REGION Network 33: **** 2.2 - Alarms - Alarms Generation **** Fuse Locc-Box Short circuit Alarm (Condition)
   // Condition for the Alarm
   #AlarmCondShortCirc := #FuseState_BitShortCirc AND #I_EnableAlarm AND NOT #C_LevelShortCirc;
END_REGION

REGION Network 34: **** 2.2 - Alarms - Alarms Generation **** Fuse Locc-Box Short circuit Alarm
   // Memorisation of the Alarm
   IF (#I_AlarmResetPB AND NOT #C_LocalResetShortCirc) OR NOT #I_EnableAlarm OR #HMICmdResetShortCirc THEN
       #AlarmShortCirc := FALSE;   // RS flip-flop
   END_IF;
   IF #AlarmCondShortCirc THEN #AlarmShortCirc := TRUE; END_IF;
END_REGION

REGION Network 35: **** 2.2 - Alarms - Alarms Generation **** Fuse Locc-Box Short circuit Warning
   // Memorisation of the Alarm
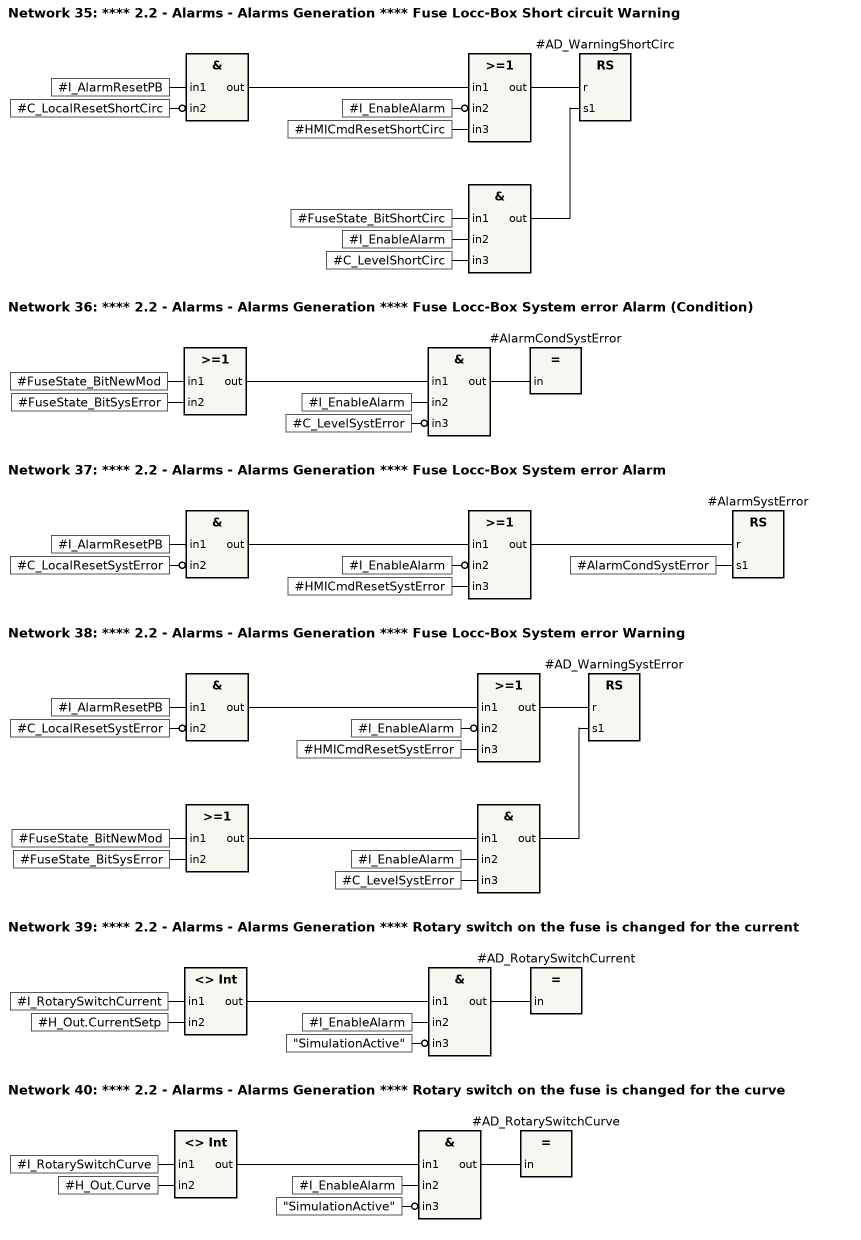
   IF (#I_AlarmResetPB AND NOT #C_LocalResetShortCirc) OR NOT #I_EnableAlarm OR #HMICmdResetShortCirc THEN
       #AD_WarningShortCirc := FALSE;   // RS flip-flop
   END_IF;
   IF #FuseState_BitShortCirc AND #I_EnableAlarm AND #C_LevelShortCirc THEN
       #AD_WarningShortCirc := TRUE;
   END_IF;
END_REGION

REGION Network 36: **** 2.2 - Alarms - Alarms Generation **** Fuse Locc-Box System error Alarm (Condition)
   // Condition for the Alarm
   #AlarmCondSystError := (#FuseState_BitNewMod OR #FuseState_BitSysError) AND #I_EnableAlarm AND NOT #C_LevelSystError;
END_REGION

REGION Network 37: **** 2.2 - Alarms - Alarms Generation **** Fuse Locc-Box System error Alarm
   // Memorisation of the Alarm
   IF (#I_AlarmResetPB AND NOT #C_LocalResetSystError) OR NOT #I_EnableAlarm OR #HMICmdResetSystError THEN
       #AlarmSystError := FALSE;   // RS flip-flop
   END_IF;
   IF #AlarmCondSystError THEN #AlarmSystError := TRUE; END_IF;
END_REGION

REGION Network 38: **** 2.2 - Alarms - Alarms Generation **** Fuse Locc-Box System error Warning
   // Memorisation of the Alarm
   IF (#I_AlarmResetPB AND NOT #C_LocalResetSystError) OR NOT #I_EnableAlarm OR #HMICmdResetSystError THEN
       #AD_WarningSystError := FALSE;   // RS flip-flop
   END_IF;
   IF (#FuseState_BitNewMod OR #FuseState_BitSysError) AND #I_EnableAlarm AND #C_LevelSystError THEN
       #AD_WarningSystError := TRUE;
   END_IF;
END_REGION

REGION Network 39: **** 2.2 - Alarms - Alarms Generation **** Rotary switch on the fuse is changed for the current
   // Alarm
   #AD_RotarySwitchCurrent := (#I_RotarySwitchCurrent <> #H_Out.CurrentSetp) AND #I_EnableAlarm AND NOT "SimulationActive";
END_REGION

REGION Network 40: **** 2.2 - Alarms - Alarms Generation **** Rotary switch on the fuse is changed for the curve
   // Alarm
   #AD_RotarySwitchCurve := (#I_RotarySwitchCurve <> #H_Out.Curve) AND #I_EnableAlarm AND NOT "SimulationActive";
END_REGION

REGION Network 41: **** 2.2 - Alarms - Alarms Generation **** Alarm = Class 'A'
   // Alarm = Class 'A'
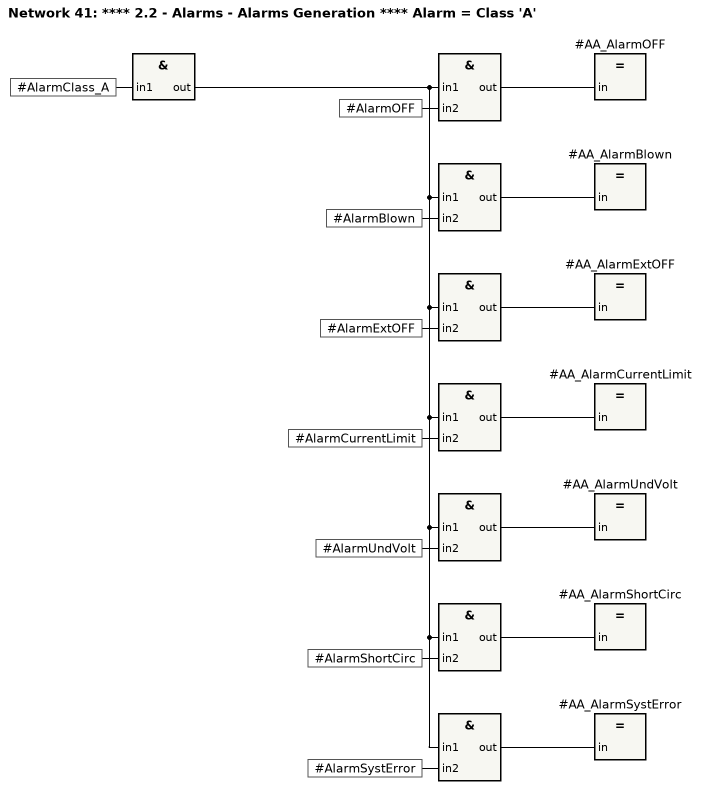
   #AA_AlarmOFF := #AlarmClass_A AND #AlarmOFF;
   #AA_AlarmBlown := #AlarmClass_A AND #AlarmBlown;
   #AA_AlarmExtOFF := #AlarmClass_A AND #AlarmExtOFF;
   #AA_AlarmCurrentLimit := #AlarmClass_A AND #AlarmCurrentLimit;
   #AA_AlarmUndVolt := #AlarmClass_A AND #AlarmUndVolt;
   #AA_AlarmShortCirc := #AlarmClass_A AND #AlarmShortCirc;
   #AA_AlarmSystError := #AlarmClass_A AND #AlarmSystError;
END_REGION

REGION Network 42: **** 2.2 - Alarms - Alarms Generation **** Alarm = Class 'B'
   // Alarm = Class 'B'
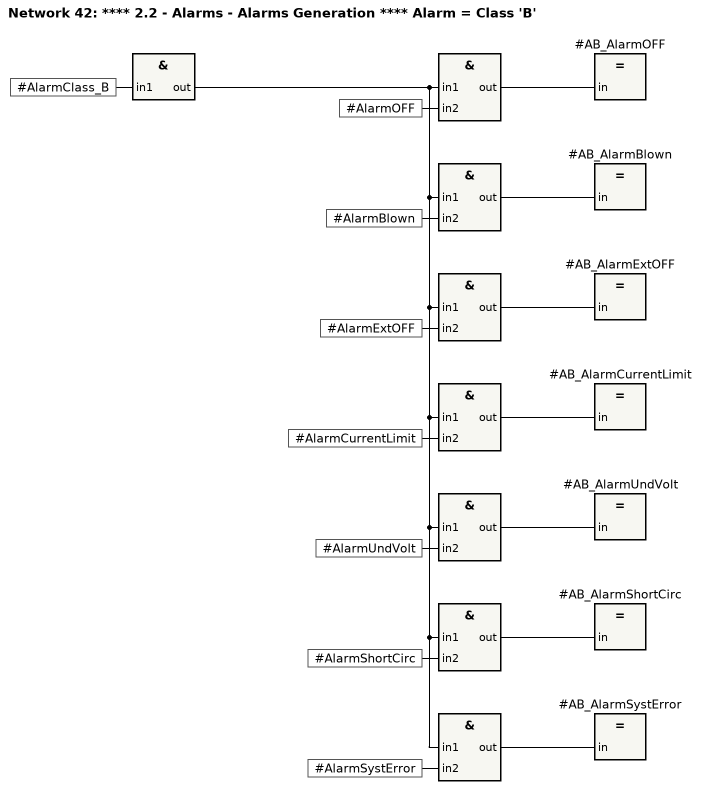
   #AB_AlarmOFF := #AlarmClass_B AND #AlarmOFF;
   #AB_AlarmBlown := #AlarmClass_B AND #AlarmBlown;
   #AB_AlarmExtOFF := #AlarmClass_B AND #AlarmExtOFF;
   #AB_AlarmCurrentLimit := #AlarmClass_B AND #AlarmCurrentLimit;
   #AB_AlarmUndVolt := #AlarmClass_B AND #AlarmUndVolt;
   #AB_AlarmShortCirc := #AlarmClass_B AND #AlarmShortCirc;
   #AB_AlarmSystError := #AlarmClass_B AND #AlarmSystError;
END_REGION

REGION Network 43: **** 2.2 - Alarms - Alarms Generation **** Alarm = Class 'C'
   // Alarm = Class 'C'
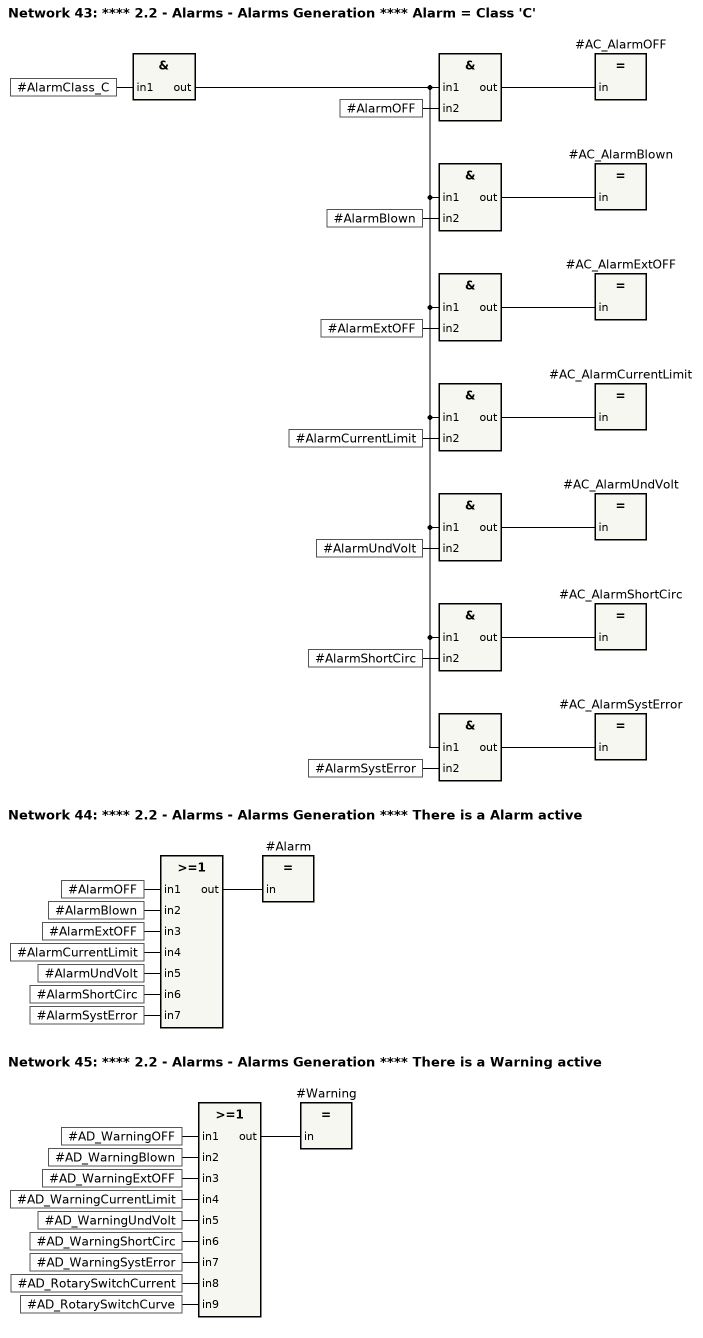
   #AC_AlarmOFF := #AlarmClass_C AND #AlarmOFF;
   #AC_AlarmBlown := #AlarmClass_C AND #AlarmBlown;
   #AC_AlarmExtOFF := #AlarmClass_C AND #AlarmExtOFF;
   #AC_AlarmCurrentLimit := #AlarmClass_C AND #AlarmCurrentLimit;
   #AC_AlarmUndVolt := #AlarmClass_C AND #AlarmUndVolt;
   #AC_AlarmShortCirc := #AlarmClass_C AND #AlarmShortCirc;
   #AC_AlarmSystError := #AlarmClass_C AND #AlarmSystError;
END_REGION

REGION Network 44: **** 2.2 - Alarms - Alarms Generation **** There is a Alarm active
   // There is a Alarm active
   #Alarm := #AlarmOFF OR #AlarmBlown OR #AlarmExtOFF OR #AlarmCurrentLimit OR #AlarmUndVolt OR #AlarmShortCirc OR #AlarmSystError;
END_REGION

REGION Network 45: **** 2.2 - Alarms - Alarms Generation **** There is a Warning active
   // There is a Warning active
   #Warning := #AD_WarningOFF OR #AD_WarningBlown OR #AD_WarningExtOFF OR #AD_WarningCurrentLimit OR #AD_WarningUndVolt OR #AD_WarningShortCirc OR #AD_WarningSystError OR #AD_RotarySwitchCurrent OR #AD_RotarySwitchCurve;
END_REGION

REGION Network 46: **** 3 - Communication - Other Systems **** Read info from LoccBox Fuse
   // Read info from LoccBox Fuse
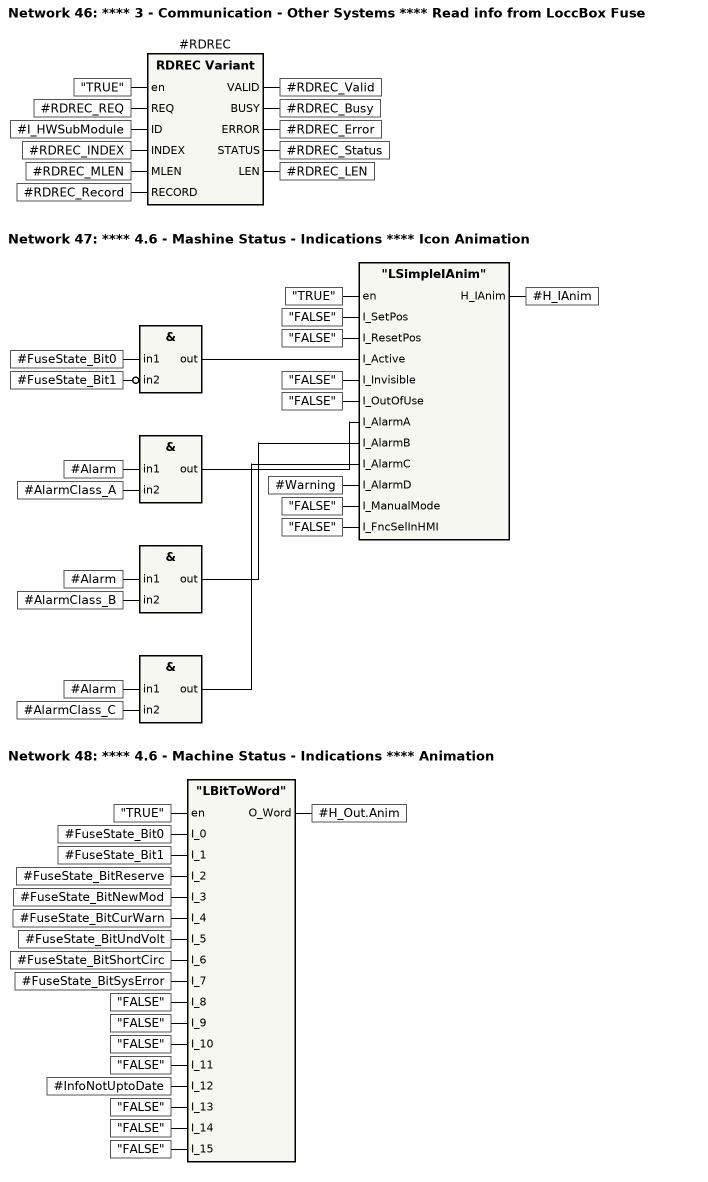
   IF "TRUE" THEN
       #RDREC(REQ := #RDREC_REQ,   // RDREC
              ID := #I_HWSubModule,
              INDEX := #RDREC_INDEX,
              MLEN := #RDREC_MLEN,
              RECORD := #RDREC_Record,
              VALID => #RDREC_Valid,
              BUSY => #RDREC_Busy,
              ERROR => #RDREC_Error,
              STATUS => #RDREC_Status,
              LEN => #RDREC_LEN);
   END_IF;
END_REGION

REGION Network 47: **** 4.6 - Mashine Status - Indications **** Icon Animation
   // Icon Animation
   IF "TRUE" THEN
       "LSimpleIAnim"(I_SetPos := "FALSE",
                      I_ResetPos := "FALSE",
                      I_Active := #FuseState_Bit0 AND NOT #FuseState_Bit1,
                      I_Invisible := "FALSE",
                      I_OutOfUse := "FALSE",
                      I_AlarmA := #Alarm AND #AlarmClass_A,
                      I_AlarmB := #Alarm AND #AlarmClass_B,
                      I_AlarmC := #Alarm AND #AlarmClass_C,
                      I_AlarmD := #Warning,
                      I_ManualMode := "FALSE",
                      I_FncSelInHMI := "FALSE",
                      H_IAnim => #H_IAnim);
   END_IF;
END_REGION

REGION Network 48: **** 4.6 - Machine Status - Indications **** Animation
   // Animation
   IF "TRUE" THEN
       "LBitToWord"(I_0 := #FuseState_Bit0,
                    I_1 := #FuseState_Bit1,
                    I_2 := #FuseState_BitReserve,
                    I_3 := #FuseState_BitNewMod,
                    I_4 := #FuseState_BitCurWarn,
                    I_5 := #FuseState_BitUndVolt,
                    I_6 := #FuseState_BitShortCirc,
                    I_7 := #FuseState_BitSysError,
                    I_8 := "FALSE",
                    I_9 := "FALSE",
                    I_10 := "FALSE",
                    I_11 := "FALSE",
                    I_12 := #InfoNotUptoDate,
                    I_13 := "FALSE",
                    I_14 := "FALSE",
                    I_15 := "FALSE",
                    O_Word => #H_Out.Anim);
   END_IF;
END_REGION

REGION Network 49: **** 4.6 - Machine Status - Indications **** Animation2
   // Animation
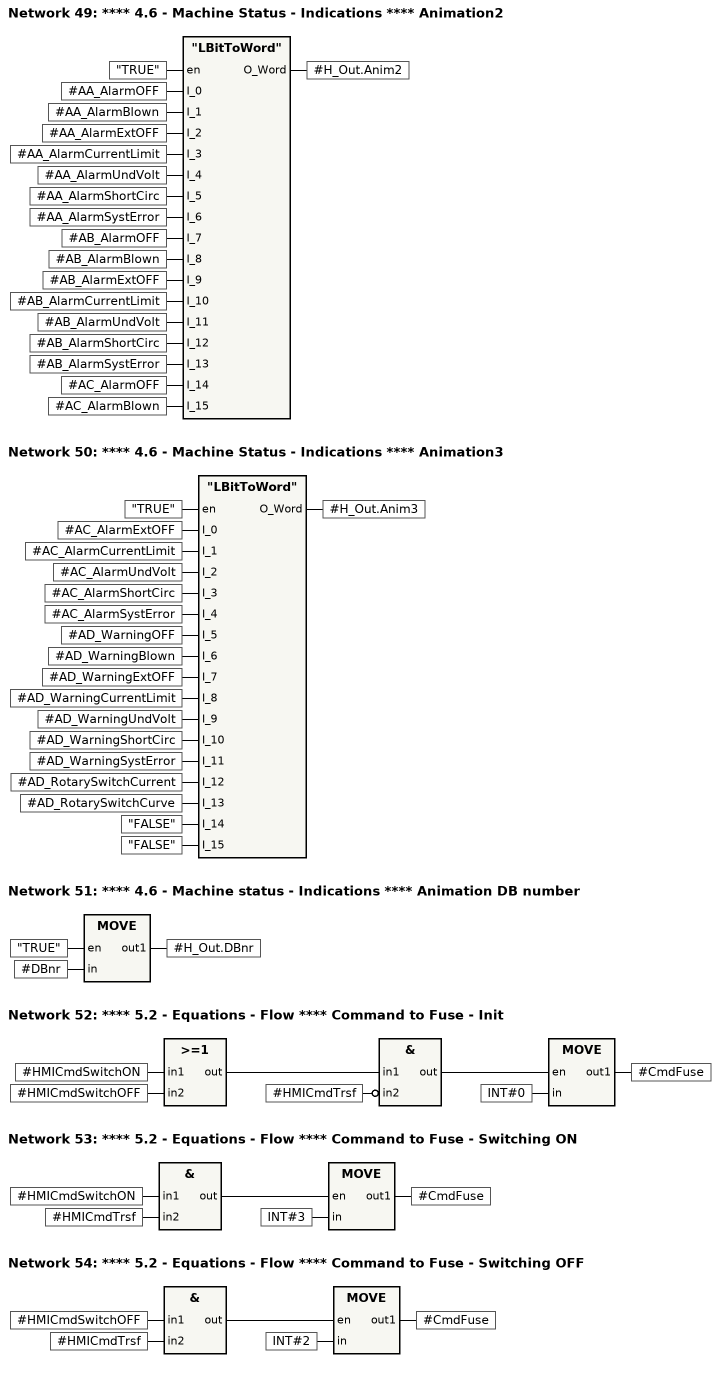
   IF "TRUE" THEN
       "LBitToWord"(I_0 := #AA_AlarmOFF,
                    I_1 := #AA_AlarmBlown,
                    I_2 := #AA_AlarmExtOFF,
                    I_3 := #AA_AlarmCurrentLimit,
                    I_4 := #AA_AlarmUndVolt,
                    I_5 := #AA_AlarmShortCirc,
                    I_6 := #AA_AlarmSystError,
                    I_7 := #AB_AlarmOFF,
                    I_8 := #AB_AlarmBlown,
                    I_9 := #AB_AlarmExtOFF,
                    I_10 := #AB_AlarmCurrentLimit,
                    I_11 := #AB_AlarmUndVolt,
                    I_12 := #AB_AlarmShortCirc,
                    I_13 := #AB_AlarmSystError,
                    I_14 := #AC_AlarmOFF,
                    I_15 := #AC_AlarmBlown,
                    O_Word => #H_Out.Anim2);
   END_IF;
END_REGION

REGION Network 50: **** 4.6 - Machine Status - Indications **** Animation3
   // Animation
   IF "TRUE" THEN
       "LBitToWord"(I_0 := #AC_AlarmExtOFF,
                    I_1 := #AC_AlarmCurrentLimit,
                    I_2 := #AC_AlarmUndVolt,
                    I_3 := #AC_AlarmShortCirc,
                    I_4 := #AC_AlarmSystError,
                    I_5 := #AD_WarningOFF,
                    I_6 := #AD_WarningBlown,
                    I_7 := #AD_WarningExtOFF,
                    I_8 := #AD_WarningCurrentLimit,
                    I_9 := #AD_WarningUndVolt,
                    I_10 := #AD_WarningShortCirc,
                    I_11 := #AD_WarningSystError,
                    I_12 := #AD_RotarySwitchCurrent,
                    I_13 := #AD_RotarySwitchCurve,
                    I_14 := "FALSE",
                    I_15 := "FALSE",
                    O_Word => #H_Out.Anim3);
   END_IF;
END_REGION

REGION Network 51: **** 4.6 - Machine status - Indications **** Animation DB number
   // DB number
   IF "TRUE" THEN #H_Out.DBnr := #DBnr; END_IF;
END_REGION

REGION Network 52: **** 5.2 - Equations - Flow **** Command to Fuse - Init
   // Write zero to outputbyte to have an transition from 0 to ...
   IF (#HMICmdSwitchON OR #HMICmdSwitchOFF) AND NOT #HMICmdTrsf THEN #CmdFuse := INT#0; END_IF;
END_REGION

REGION Network 53: **** 5.2 - Equations - Flow **** Command to Fuse - Switching ON
   // Switching ON
   IF #HMICmdSwitchON AND #HMICmdTrsf THEN #CmdFuse := INT#3; END_IF;
END_REGION

REGION Network 54: **** 5.2 - Equations - Flow **** Command to Fuse - Switching OFF
   // Switching OFF
   IF #HMICmdSwitchOFF AND #HMICmdTrsf THEN #CmdFuse := INT#2; END_IF;
END_REGION

REGION Network 55: **** 5.2 - Equations - Flow **** Start Read function (GET Info)
   // Start Read function
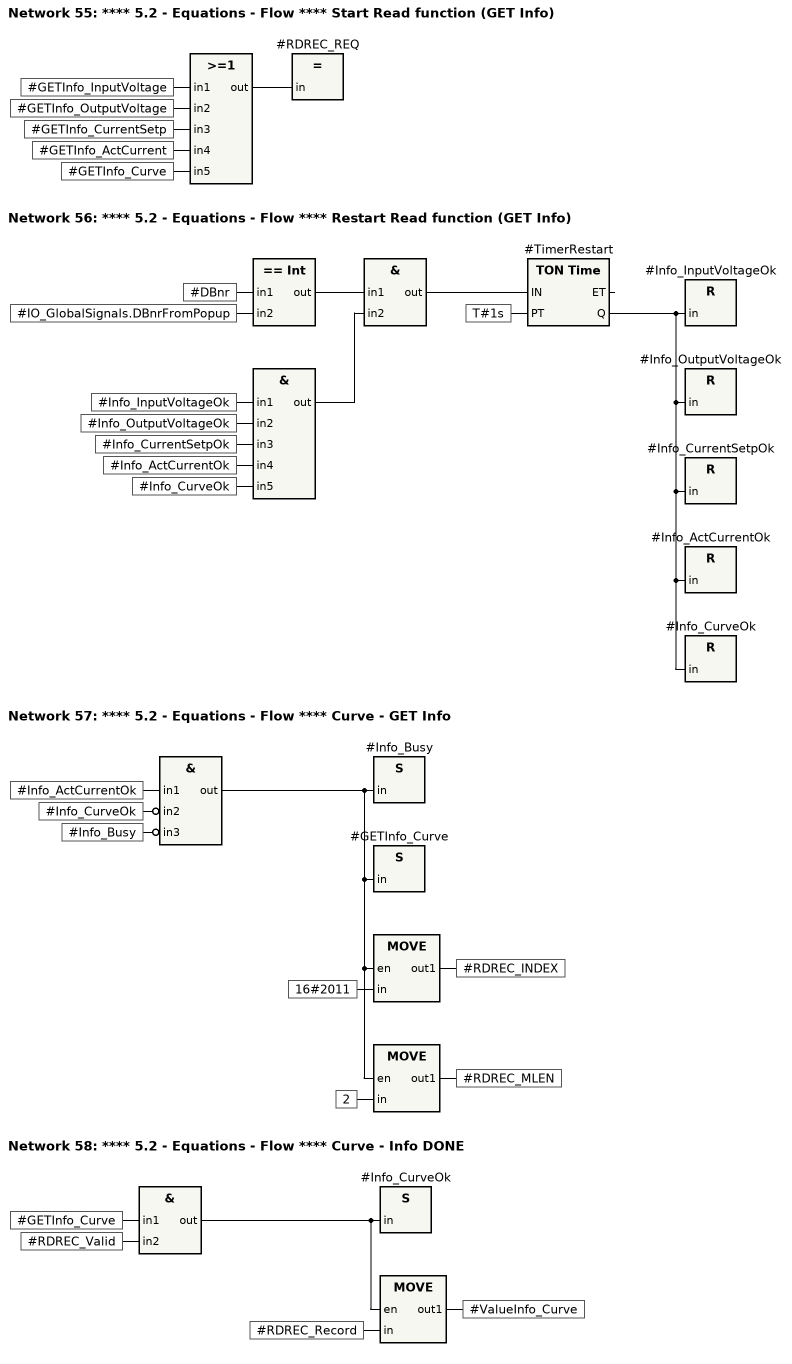
   #RDREC_REQ := #GETInfo_InputVoltage OR #GETInfo_OutputVoltage OR #GETInfo_CurrentSetp OR #GETInfo_ActCurrent OR #GETInfo_Curve;
END_REGION

REGION Network 56: **** 5.2 - Equations - Flow **** Restart Read function (GET Info)
   // Restart Read function (GET Info)
   #TimerRestart(IN := (#DBnr = #IO_GlobalSignals.DBnrFromPopup) AND #Info_InputVoltageOk AND #Info_OutputVoltageOk AND #Info_CurrentSetpOk AND #Info_ActCurrentOk AND #Info_CurveOk,   // TON
                 PT := T#1s);
   IF #TimerRestart.Q THEN
       #Info_InputVoltageOk := FALSE;
       #Info_OutputVoltageOk := FALSE;
       #Info_CurrentSetpOk := FALSE;
       #Info_ActCurrentOk := FALSE;
       #Info_CurveOk := FALSE;
   END_IF;
END_REGION

REGION Network 57: **** 5.2 - Equations - Flow **** Curve - GET Info
   // GET Info Curve
   #_w1 := #Info_ActCurrentOk AND NOT #Info_CurveOk AND NOT #Info_Busy;
   IF #_w1 THEN
       #Info_Busy := TRUE;
       #GETInfo_Curve := TRUE;
       #RDREC_INDEX := 16#2011;
       #RDREC_MLEN := 2;
   END_IF;
END_REGION

REGION Network 58: **** 5.2 - Equations - Flow **** Curve - Info DONE
   // DONE Info Curve
   IF #GETInfo_Curve AND #RDREC_Valid THEN
       #Info_CurveOk := TRUE;
       #ValueInfo_Curve := #RDREC_Record;
   END_IF;
END_REGION

REGION Network 59: **** 5.2 - Equations - Flow **** Curve - CALCULATE
   // CALCULATE Current Curve
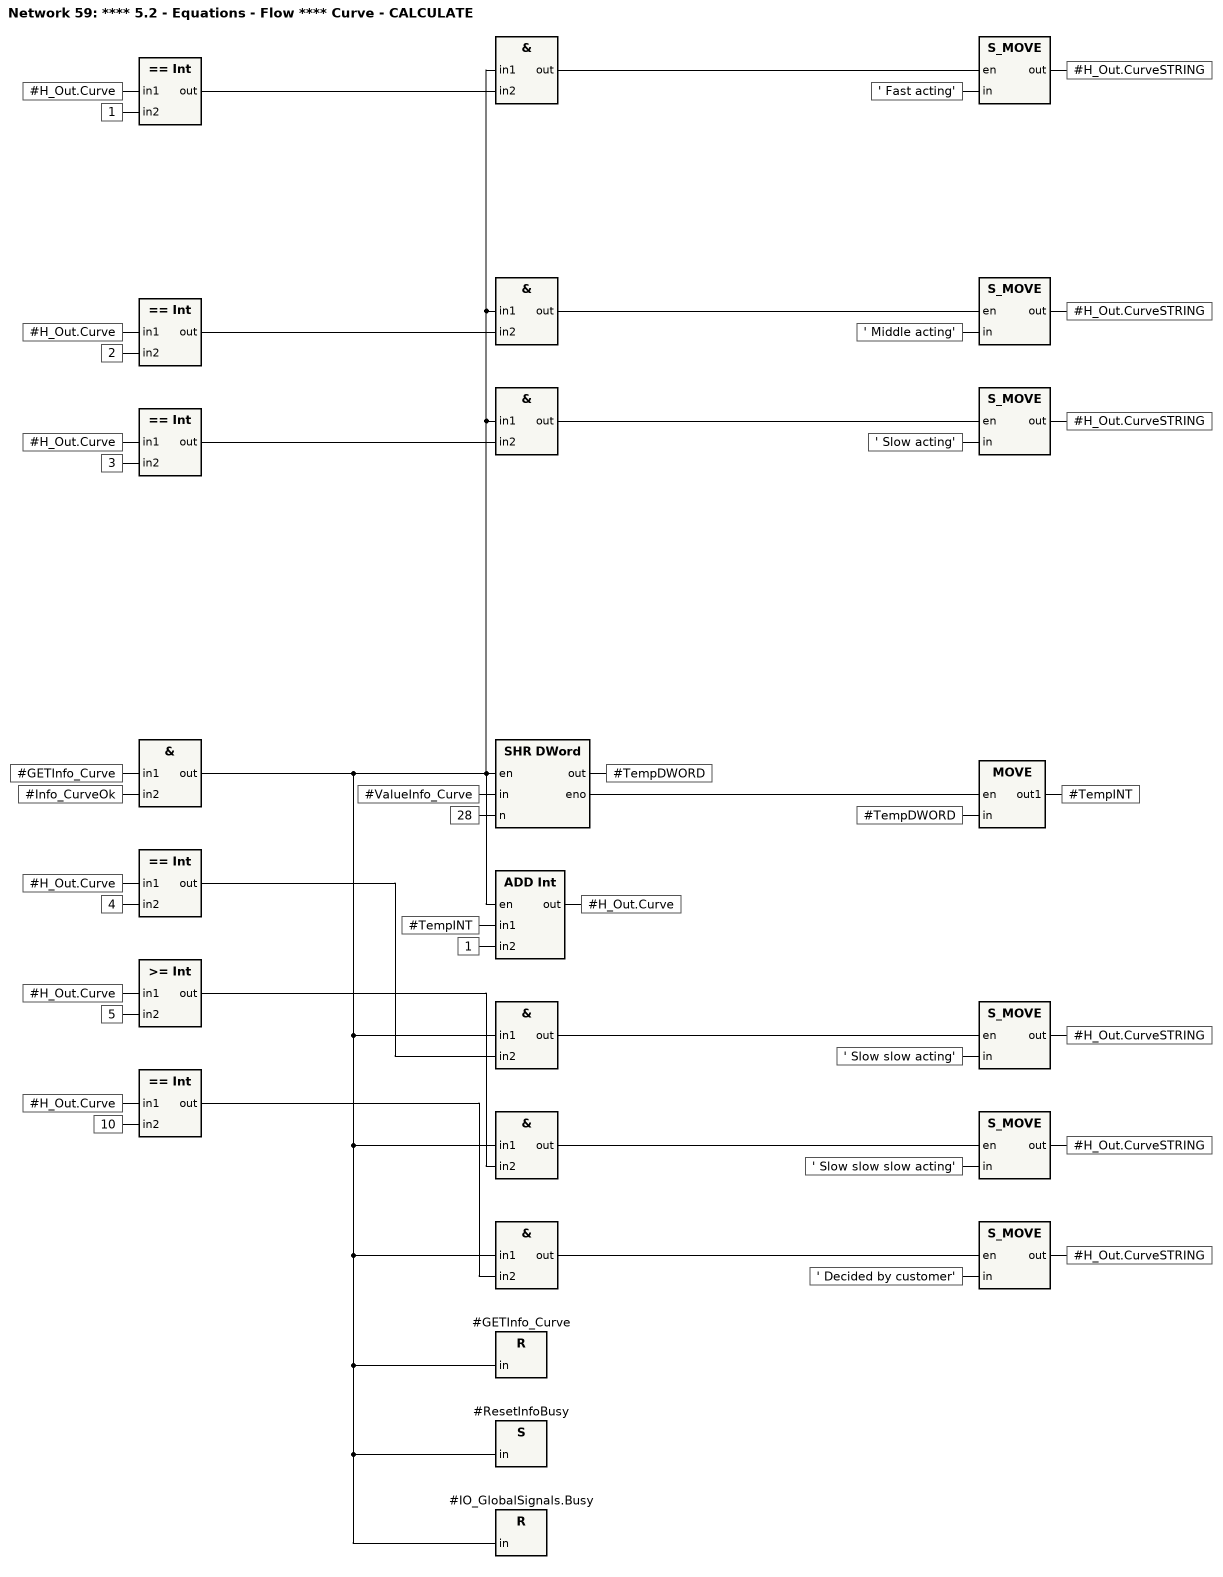
   #_w1 := #GETInfo_Curve AND #Info_CurveOk;
   IF #_w1 THEN
       #TempDWORD := SHR(IN := #ValueInfo_Curve, N := 28);
       #TempINT := #TempDWORD;
       #H_Out.Curve := #TempINT + 1;
   END_IF;
   IF #_w1 AND (#H_Out.Curve = 1) THEN #H_Out.CurveSTRING := ' Fast acting'; END_IF;
   IF #_w1 AND (#H_Out.Curve = 2) THEN #H_Out.CurveSTRING := ' Middle acting'; END_IF;
   IF #_w1 AND (#H_Out.Curve = 3) THEN #H_Out.CurveSTRING := ' Slow acting'; END_IF;
   IF #_w1 AND (#H_Out.Curve = 4) THEN #H_Out.CurveSTRING := ' Slow slow acting'; END_IF;
   IF #_w1 AND (#H_Out.Curve >= 5) THEN #H_Out.CurveSTRING := ' Slow slow slow acting'; END_IF;
   IF #_w1 AND (#H_Out.Curve = 10) THEN #H_Out.CurveSTRING := ' Decided by customer'; END_IF;
   IF #_w1 THEN
       #GETInfo_Curve := FALSE;
       #ResetInfoBusy := TRUE;
       #IO_GlobalSignals.Busy := FALSE;
   END_IF;
END_REGION

REGION Network 60: **** 5.2 - Equations - Flow **** Actual Current - GET Info
   // GET Info Actual Current
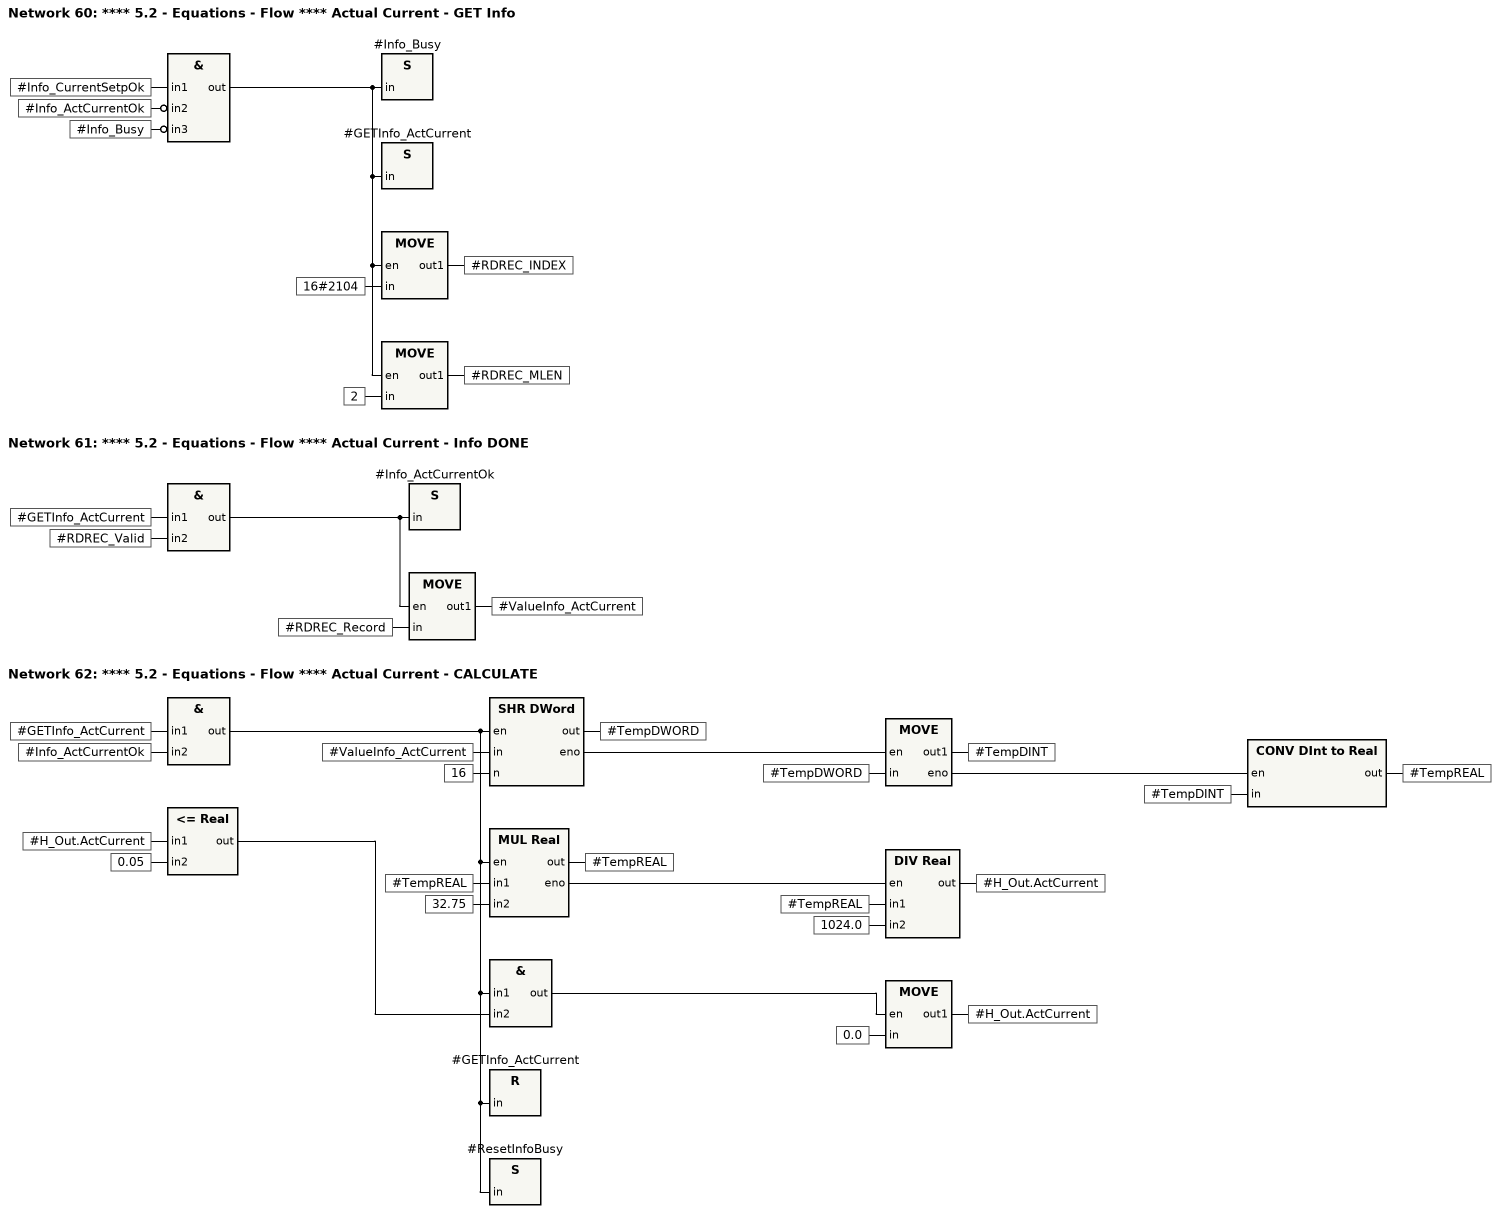
   #_w1 := #Info_CurrentSetpOk AND NOT #Info_ActCurrentOk AND NOT #Info_Busy;
   IF #_w1 THEN
       #Info_Busy := TRUE;
       #GETInfo_ActCurrent := TRUE;
       #RDREC_INDEX := 16#2104;
       #RDREC_MLEN := 2;
   END_IF;
END_REGION

REGION Network 61: **** 5.2 - Equations - Flow **** Actual Current - Info DONE
   // DONE Info Actual Current
   IF #GETInfo_ActCurrent AND #RDREC_Valid THEN
       #Info_ActCurrentOk := TRUE;
       #ValueInfo_ActCurrent := #RDREC_Record;
   END_IF;
END_REGION

REGION Network 62: **** 5.2 - Equations - Flow **** Actual Current - CALCULATE
   // CALCULATE Actual Current   ----->  Actual Current = (ValueInfo_ActCurrent * 32,75A) / 1024
   #_w1 := #GETInfo_ActCurrent AND #Info_ActCurrentOk;
   IF #_w1 THEN
       #TempDWORD := SHR(IN := #ValueInfo_ActCurrent, N := 16);
       #TempDINT := #TempDWORD;
       #TempREAL := DINT_TO_REAL(#TempDINT);
       #TempREAL := #TempREAL * 32.75;
       #H_Out.ActCurrent := #TempREAL / 1024.0;
   END_IF;
   IF #_w1 AND (#H_Out.ActCurrent <= 0.05) THEN #H_Out.ActCurrent := 0.0; END_IF;
   IF #_w1 THEN
       #GETInfo_ActCurrent := FALSE;
       #ResetInfoBusy := TRUE;
   END_IF;
END_REGION

REGION Network 63: **** 5.2 - Equations - Flow **** Current Setpoint - GET Info
   // GET Info Current Setpoint
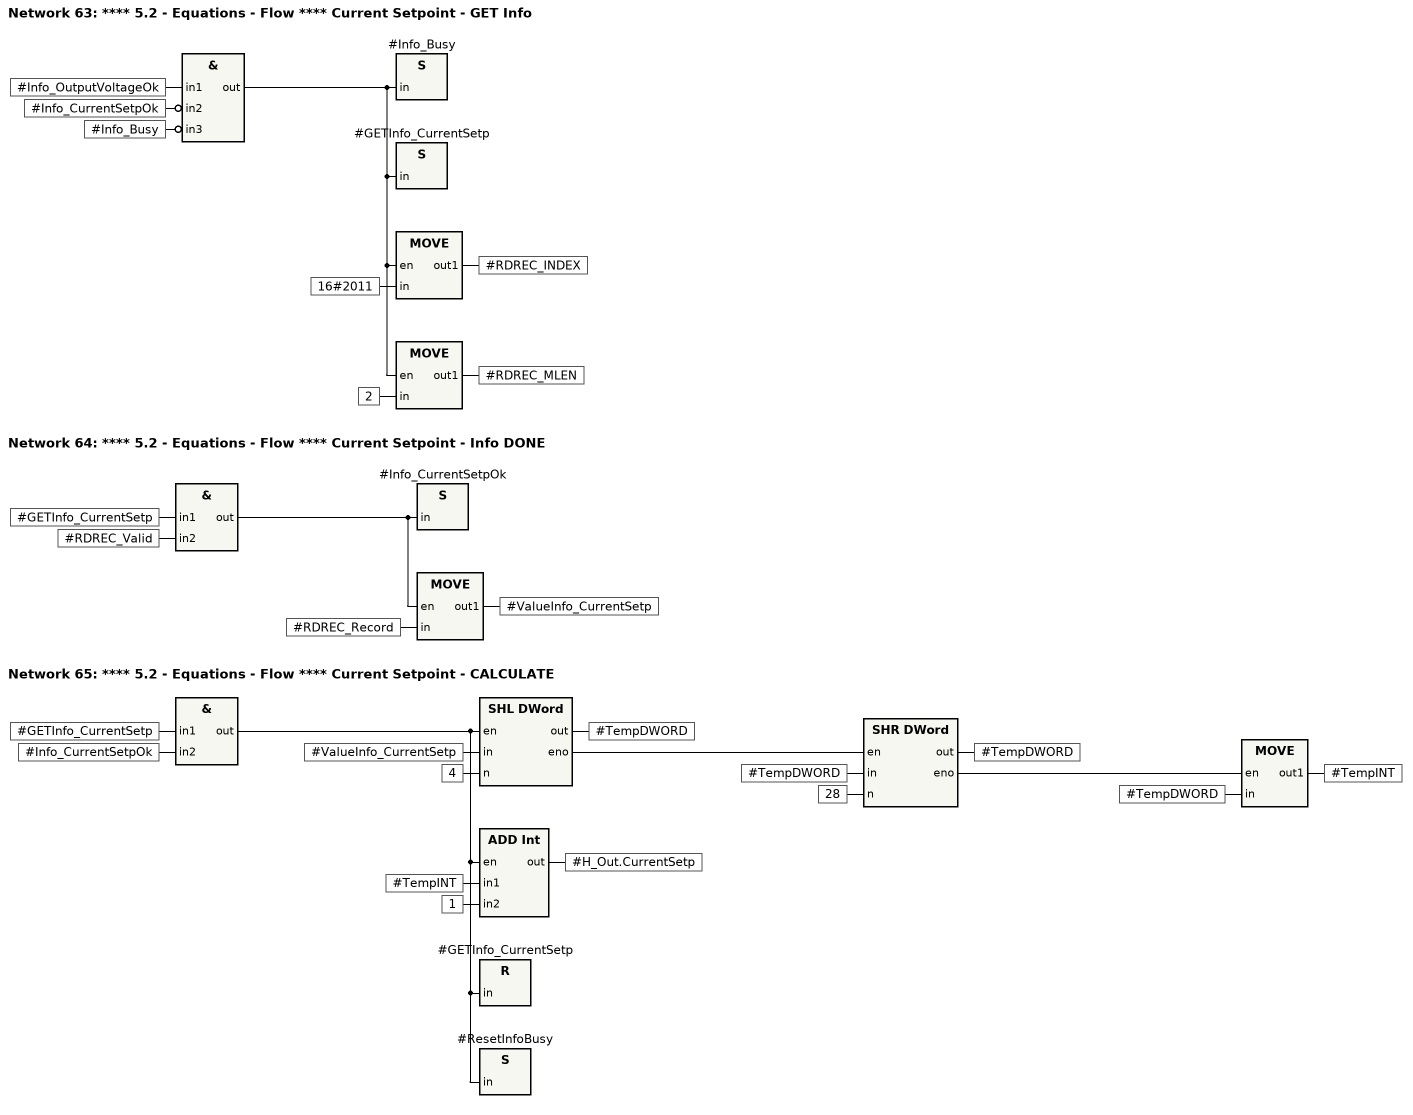
   #_w1 := #Info_OutputVoltageOk AND NOT #Info_CurrentSetpOk AND NOT #Info_Busy;
   IF #_w1 THEN
       #Info_Busy := TRUE;
       #GETInfo_CurrentSetp := TRUE;
       #RDREC_INDEX := 16#2011;
       #RDREC_MLEN := 2;
   END_IF;
END_REGION

REGION Network 64: **** 5.2 - Equations - Flow **** Current Setpoint - Info DONE
   // DONE Info Current Setpoint
   IF #GETInfo_CurrentSetp AND #RDREC_Valid THEN
       #Info_CurrentSetpOk := TRUE;
       #ValueInfo_CurrentSetp := #RDREC_Record;
   END_IF;
END_REGION

REGION Network 65: **** 5.2 - Equations - Flow **** Current Setpoint - CALCULATE
   // CALCULATE Current Setpoint
   IF #GETInfo_CurrentSetp AND #Info_CurrentSetpOk THEN
       #TempDWORD := SHL(IN := #ValueInfo_CurrentSetp, N := 4);
       #TempDWORD := SHR(IN := #TempDWORD, N := 28);
       #TempINT := #TempDWORD;
       #H_Out.CurrentSetp := #TempINT + 1;
   END_IF;
   #_w1 := #GETInfo_CurrentSetp AND #Info_CurrentSetpOk;
   IF #_w1 THEN
       #GETInfo_CurrentSetp := FALSE;
       #ResetInfoBusy := TRUE;
   END_IF;
END_REGION

REGION Network 66: **** 5.2 - Equations - Flow **** Output Voltage - GET Info
   // GET Info Output Voltage
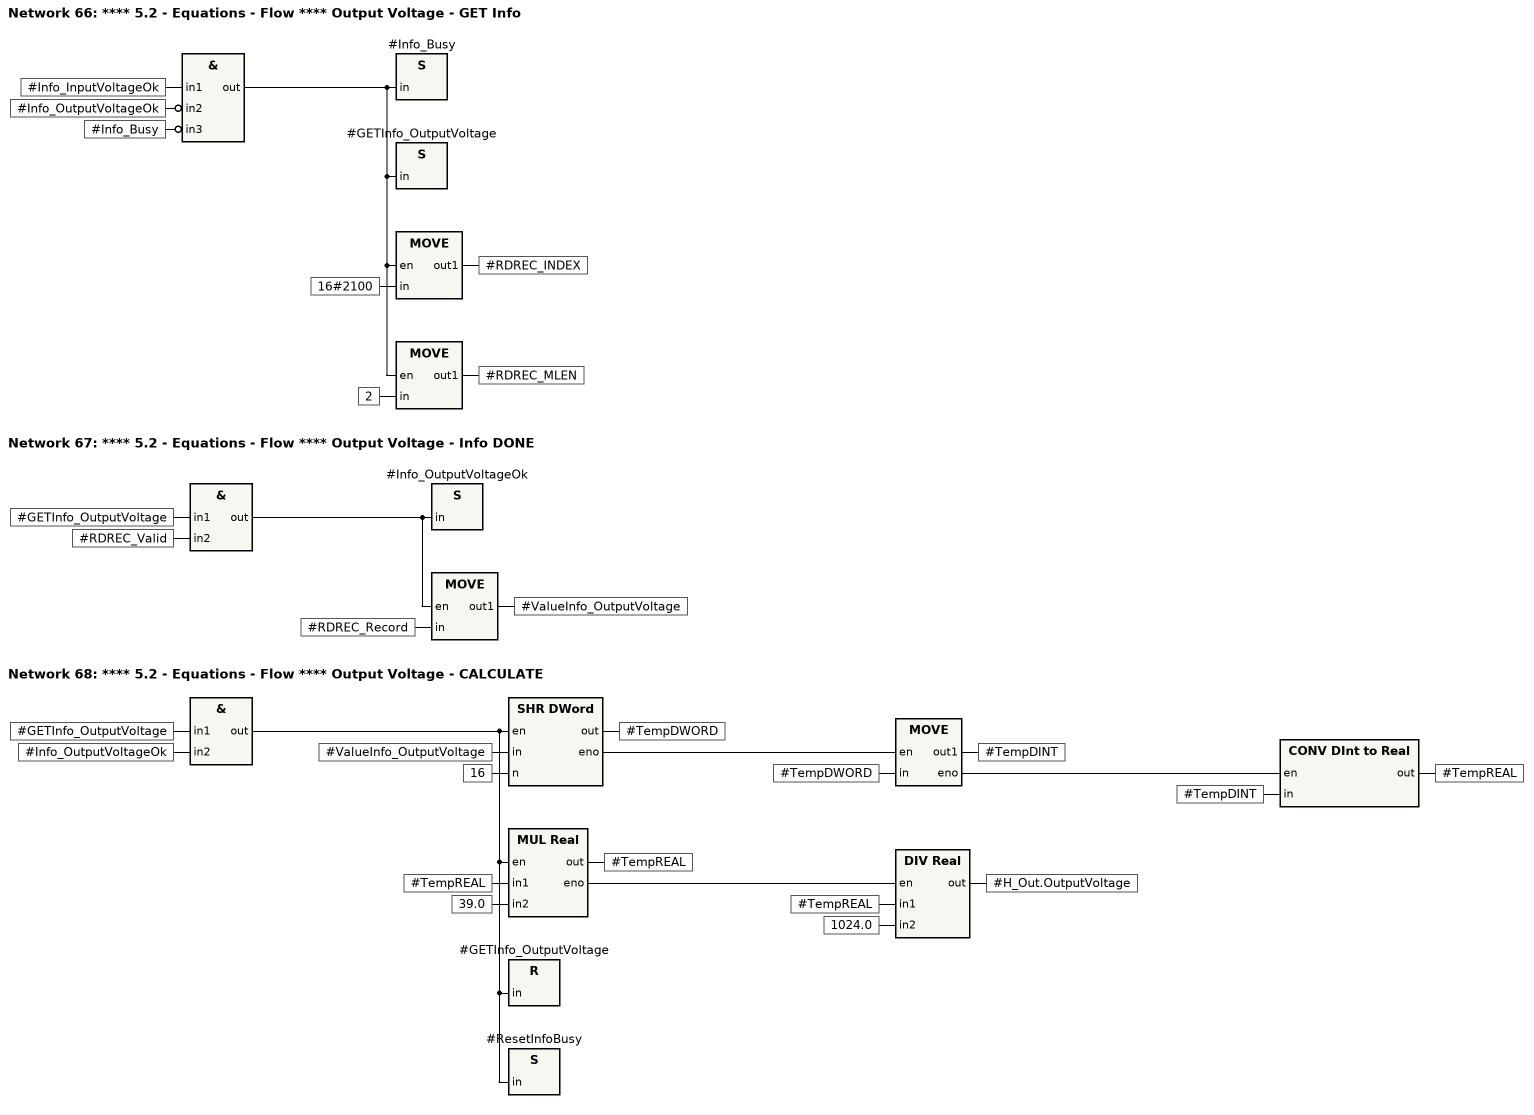
   #_w1 := #Info_InputVoltageOk AND NOT #Info_OutputVoltageOk AND NOT #Info_Busy;
   IF #_w1 THEN
       #Info_Busy := TRUE;
       #GETInfo_OutputVoltage := TRUE;
       #RDREC_INDEX := 16#2100;
       #RDREC_MLEN := 2;
   END_IF;
END_REGION

REGION Network 67: **** 5.2 - Equations - Flow **** Output Voltage - Info DONE
   // DONE Info Output Voltage
   IF #GETInfo_OutputVoltage AND #RDREC_Valid THEN
       #Info_OutputVoltageOk := TRUE;
       #ValueInfo_OutputVoltage := #RDREC_Record;
   END_IF;
END_REGION

REGION Network 68: **** 5.2 - Equations - Flow **** Output Voltage - CALCULATE
   // CALCULATE Output Voltage   ----->  Output Voltage = (ValueInfo_OutputVoltage * 39V) / 1024
   IF #GETInfo_OutputVoltage AND #Info_OutputVoltageOk THEN
       #TempDWORD := SHR(IN := #ValueInfo_OutputVoltage, N := 16);
       #TempDINT := #TempDWORD;
       #TempREAL := DINT_TO_REAL(#TempDINT);
       #TempREAL := #TempREAL * 39.0;
       #H_Out.OutputVoltage := #TempREAL / 1024.0;
   END_IF;
   #_w1 := #GETInfo_OutputVoltage AND #Info_OutputVoltageOk;
   IF #_w1 THEN
       #GETInfo_OutputVoltage := FALSE;
       #ResetInfoBusy := TRUE;
   END_IF;
END_REGION

REGION Network 69: **** 5.2 - Equations - Flow **** Input Voltage - GET Info
   // GET Info Input Voltage
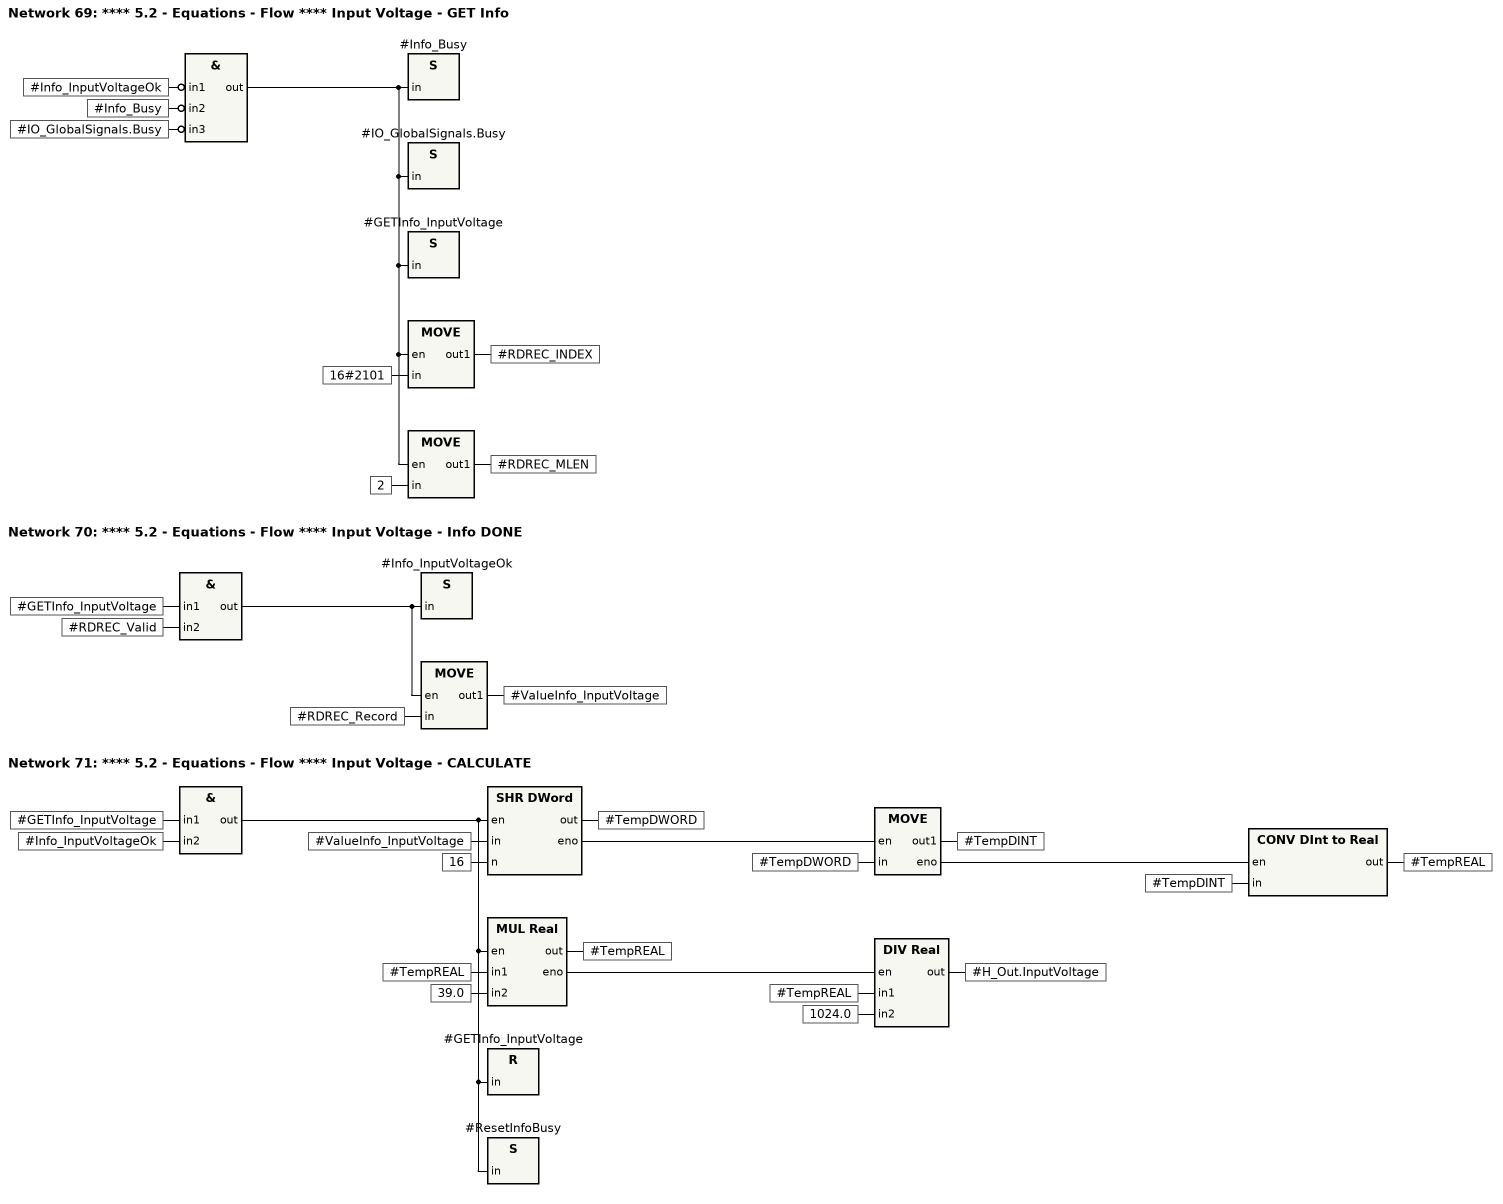
   #_w1 := NOT #Info_InputVoltageOk AND NOT #Info_Busy AND NOT #IO_GlobalSignals.Busy;
   IF #_w1 THEN
       #Info_Busy := TRUE;
       #IO_GlobalSignals.Busy := TRUE;
       #GETInfo_InputVoltage := TRUE;
       #RDREC_INDEX := 16#2101;
       #RDREC_MLEN := 2;
   END_IF;
END_REGION

REGION Network 70: **** 5.2 - Equations - Flow **** Input Voltage - Info DONE
   // DONE Info Input Voltage
   IF #GETInfo_InputVoltage AND #RDREC_Valid THEN
       #Info_InputVoltageOk := TRUE;
       #ValueInfo_InputVoltage := #RDREC_Record;
   END_IF;
END_REGION

REGION Network 71: **** 5.2 - Equations - Flow **** Input Voltage - CALCULATE
   // CALCULATE Input Voltage   ----->  Input Voltage = (ValueInfo_InputVoltage * 39V) / 1024
   IF #GETInfo_InputVoltage AND #Info_InputVoltageOk THEN
       #TempDWORD := SHR(IN := #ValueInfo_InputVoltage, N := 16);
       #TempDINT := #TempDWORD;
       #TempREAL := DINT_TO_REAL(#TempDINT);
       #TempREAL := #TempREAL * 39.0;
       #H_Out.InputVoltage := #TempREAL / 1024.0;
   END_IF;
   #_w1 := #GETInfo_InputVoltage AND #Info_InputVoltageOk;
   IF #_w1 THEN
       #GETInfo_InputVoltage := FALSE;
       #ResetInfoBusy := TRUE;
   END_IF;
END_REGION

REGION Network 72: **** 5.2 - Equations - Flow **** Local Busy
   // Local Busy
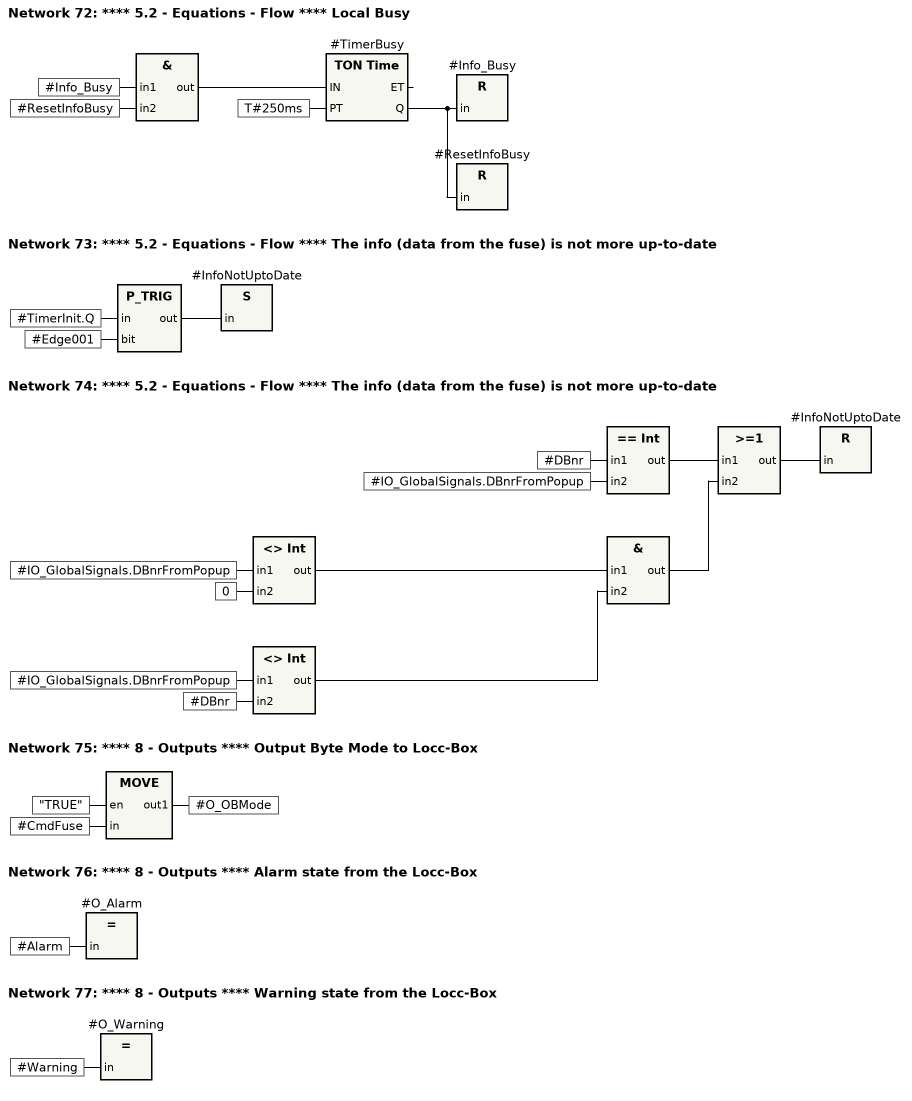
   #TimerBusy(IN := #Info_Busy AND #ResetInfoBusy, PT := T#250ms);   // TON
   IF #TimerBusy.Q THEN
       #Info_Busy := FALSE;
       #ResetInfoBusy := FALSE;
   END_IF;
END_REGION

REGION Network 73: **** 5.2 - Equations - Flow **** The info (data from the fuse) is not more up-to-date
   // The info (data from the fuse) is not more up-to-date
   #_w1 := #TimerInit.Q AND NOT #Edge001;   // rising edge
   #Edge001 := #TimerInit.Q;
   IF #_w1 THEN #InfoNotUptoDate := TRUE; END_IF;
END_REGION

REGION Network 74: **** 5.2 - Equations - Flow **** The info (data from the fuse) is not more up-to-date
   // The info (data from the fuse) is not more up-to-date
   IF (#DBnr = #IO_GlobalSignals.DBnrFromPopup) OR ((#IO_GlobalSignals.DBnrFromPopup <> 0) AND (#IO_GlobalSignals.DBnrFromPopup <> #DBnr)) THEN
       #InfoNotUptoDate := FALSE;
   END_IF;
END_REGION

REGION Network 75: **** 8 - Outputs **** Output Byte Mode to Locc-Box
   // Output Byte Mode to Locc-Box
   IF "TRUE" THEN #O_OBMode := #CmdFuse; END_IF;
END_REGION

REGION Network 76: **** 8 - Outputs **** Alarm state from the Locc-Box
   // Alarm state from the Locc-Box
   #O_Alarm := #Alarm;
END_REGION

REGION Network 77: **** 8 - Outputs **** Warning state from the Locc-Box
   // Warning state from the Locc-Box
   #O_Warning := #Warning;
END_REGION

REGION Network 78: **** 8 - Outputs **** Alarm AB condition
   // Alarm AB condition
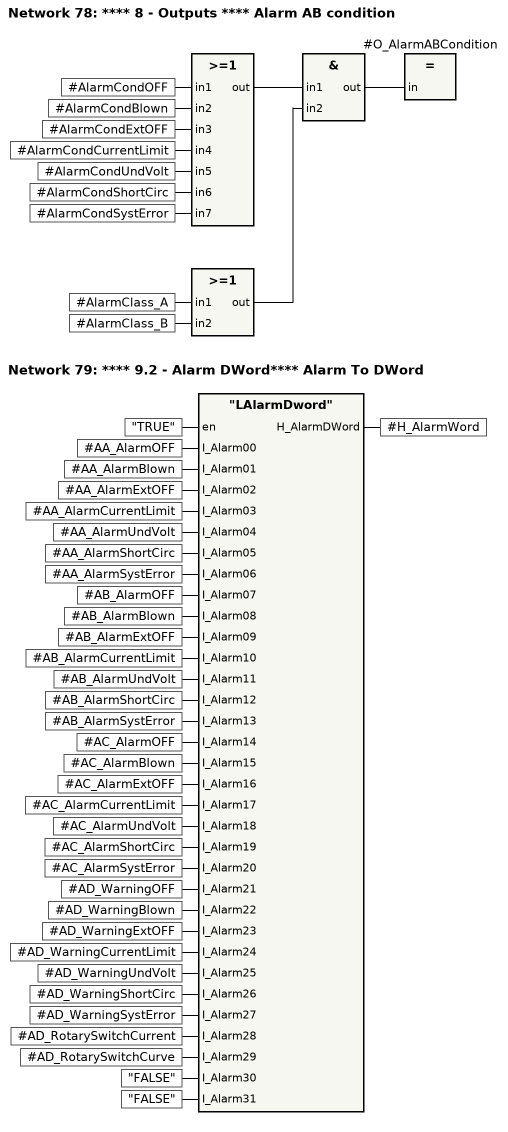
   #O_AlarmABCondition := (#AlarmCondOFF OR #AlarmCondBlown OR #AlarmCondExtOFF OR #AlarmCondCurrentLimit OR #AlarmCondUndVolt OR #AlarmCondShortCirc OR #AlarmCondSystError) AND (#AlarmClass_A OR #AlarmClass_B);
END_REGION

REGION Network 79: **** 9.2 - Alarm DWord**** Alarm To DWord
   // Alarm Word
   IF "TRUE" THEN
       "LAlarmDword"(I_Alarm00 := #AA_AlarmOFF,
                     I_Alarm01 := #AA_AlarmBlown,
                     I_Alarm02 := #AA_AlarmExtOFF,
                     I_Alarm03 := #AA_AlarmCurrentLimit,
                     I_Alarm04 := #AA_AlarmUndVolt,
                     I_Alarm05 := #AA_AlarmShortCirc,
                     I_Alarm06 := #AA_AlarmSystError,
                     I_Alarm07 := #AB_AlarmOFF,
                     I_Alarm08 := #AB_AlarmBlown,
                     I_Alarm09 := #AB_AlarmExtOFF,
                     I_Alarm10 := #AB_AlarmCurrentLimit,
                     I_Alarm11 := #AB_AlarmUndVolt,
                     I_Alarm12 := #AB_AlarmShortCirc,
                     I_Alarm13 := #AB_AlarmSystError,
                     I_Alarm14 := #AC_AlarmOFF,
                     I_Alarm15 := #AC_AlarmBlown,
                     I_Alarm16 := #AC_AlarmExtOFF,
                     I_Alarm17 := #AC_AlarmCurrentLimit,
                     I_Alarm18 := #AC_AlarmUndVolt,
                     I_Alarm19 := #AC_AlarmShortCirc,
                     I_Alarm20 := #AC_AlarmSystError,
                     I_Alarm21 := #AD_WarningOFF,
                     I_Alarm22 := #AD_WarningBlown,
                     I_Alarm23 := #AD_WarningExtOFF,
                     I_Alarm24 := #AD_WarningCurrentLimit,
                     I_Alarm25 := #AD_WarningUndVolt,
                     I_Alarm26 := #AD_WarningShortCirc,
                     I_Alarm27 := #AD_WarningSystError,
                     I_Alarm28 := #AD_RotarySwitchCurrent,
                     I_Alarm29 := #AD_RotarySwitchCurve,
                     I_Alarm30 := "FALSE",
                     I_Alarm31 := "FALSE",
                     H_AlarmDWord => #H_AlarmWord);
   END_IF;
END_REGION
END_FUNCTION_BLOCK

FUNCTION_BLOCK "LETAFuseAlarm"   // FB1413, FBD
TITLE = LLoccBoxAlarm / LETAFuseAlarm
{ S7_Optimized_Access := 'FALSE' }
AUTHOR : VCG
FAMILY : AlarmHnd
NAME : SpcGB
VERSION : 1.0
// ================================================================================
// This module is used for installations with Locc-Box type 7-6410.
// It create alarms and warning in function of configuration and status from the 
// Box.
// It Send Mode byte to the Box in function of Pop-up and external commands
// ================================================================================
// C_AlarmOrWarning
// Bit0: C_LevelOFF (Bit ON=Warning ; OFF=Alarm)
// Bit1: C_LevelBlown (Bit ON=Warning ; OFF=Alarm)
// Bit2: C_LevelExtOFF (Bit ON=Warning ; OFF=Alarm)
// Bit3: C_LevelCurrentLimit (Bit ON=Warning ; OFF=Alarm)
// Bit4: C_LevelUndVolt (Bit ON=Warning ; OFF=Alarm)
// Bit5: C_LevelShortCirc (Bit ON=Warning ; OFF=Alarm)
// Bit6: C_LevelSystError (Bit ON=Warning ; OFF=Alarm)
// Bit7: C_LevelSpareBit7
// Bit8: C_LevelSpareBit8
// Bit9: C_LevelSpareBit9
// Bit10:C_LevelSpareBit10
// Bit11:C_LevelSpareBit11
// Bit12:C_LevelSpareBit12
// Bit13:C_LevelSpareBit13
// Bit14:C_LevelSpareBit14
// Bit15:C_LevelSpareBit15
// ================================================================================
// H_HMICmd
// Bit0: HMICmdSwitchON (Bit PosEdge = Request ON)
// Bit1: HMICmdSwitchOFF (Bit PosEdge = Request OFF)
// Bit2: HMICmdResetOFF (Bit PosEdge = Reset OFF)
// Bit3: HMICmdResetExtOFF (Bit PosEdge = Reset ExtOFF)
// Bit4: HMICmdResetCurrentLimit(Bit PosEdge = Reset CurrentLimit)
// Bit5: HMICmdResetUndVolt(Bit PosEdge = Reset UndVolt)
// Bit6: HMICmdResetShortCirc(Bit PosEdge = Reset ShortCirc)
// Bit7: HMICmdResetSystError(Bit PosEdge = Reset SystError)
// Bit8: HMICmdSpareBit8
// Bit9: HMICmdSpareBit9
// Bit10:HMICmdSpareBit10
// Bit11:HMICmdSpareBit11
// Bit12:HMICmdSpareBit12
// Bit13:HMICmdSpareBit13
// Bit14:HMICmdSpareBit14
// Bit15:HMICmdSpareBit15
// ================================================================================
// C_LocalOrRemoteReset
// Bit0: C_LocalResetOFF (Bit ON=LocalResetOnly ; OFF=RemoteResetPossible)
// Bit1: C_LocalResetBlown (Bit ON=LocalResetOnly ; OFF=RemoteResetPossible)
// Bit2: C_LocalResetExtOFF (Bit ON=LocalResetOnly ; OFF=RemoteResetPossible)
// Bit3: C_LocalResetCurrentLimit (Bit ON=LocalResetOnly ; OFF=RemoteResetPossible)
// Bit4: C_LocalResetUndVolt (Bit ON=LocalResetOnly ; OFF=RemoteResetPossible)
// Bit5: C_LocalResetShortCirc (Bit ON=LocalResetOnly ; OFF=RemoteResetPossible)
// Bit6: C_LocalResetSystError (Bit ON=LocalResetOnly ; OFF=RemoteResetPossible)
// Bit7: C_LocalResetBit7
// Bit8: C_LocalResetBit8
// Bit9: C_LocalResetBit9
// Bit10:C_LocalResetBit10
// Bit11:C_LocalResetBit11
// Bit12:C_LocalResetBit12
// Bit13:C_LocalResetBit13
// Bit14:C_LocalResetBit14
// Bit15:C_LocalResetBit15
// 
// Updated to make fuse resetable from WinCC (Through HMI cmd)
// stored: AutoNumber false, IsIECCheckEnabled false, SetENOAutomatically False, UDAEnableTagReadback false
   VAR_INPUT
      I_AlarmClass { ExternalAccessible := 'False'; ExternalVisible := 'False'; ExternalWritable := 'False'} : Char;   // Alarm class -> A - B or C / Alarm class -> A - B - C or D
      I_EnableAlarm { ExternalAccessible := 'False'; ExternalVisible := 'False'; ExternalWritable := 'False'} : Bool := TRUE;   // Enable alarm from upper level
      I_AlarmResetPB { ExternalAccessible := 'False'; ExternalVisible := 'False'; ExternalWritable := 'False'} : Bool;   // Alarm reset pushbutton is activated
      C_AlarmOrWarning { ExternalAccessible := 'False'; ExternalVisible := 'False'; ExternalWritable := 'False'} : Word;   // Used to define if for this installation a status is alarm or warning
      C_LocalOrRemoteReset { ExternalAccessible := 'False'; ExternalVisible := 'False'; ExternalWritable := 'False'} : Word;   // Used to define if for this installation an error is local or remote reset
      C_Config { ExternalAccessible := 'False'; ExternalVisible := 'False'; ExternalWritable := 'False'} : "ETAFuseCPC20PNConfig";   // Config
   END_VAR
   VAR_OUTPUT
      O_Alarm { ExternalAccessible := 'False'; ExternalVisible := 'False'; ExternalWritable := 'False'} : Bool;   // Alarm state from the Locc-Box (Alarm list done inside) / Alarm state from the ETA Fuse (Alarm list done inside)
      O_Warning { ExternalAccessible := 'False'; ExternalVisible := 'False'; ExternalWritable := 'False'} : Bool;   // Warning state from the Locc-Box (Alarm list done inside) / Warning state from the ETA Fuse (Alarm list done inside)
      O_AlarmABCondition { ExternalAccessible := 'False'; ExternalVisible := 'False'; ExternalWritable := 'False'} : Bool;   // Alarm AB condition
      H_IAnim { ExternalAccessible := 'False'; ExternalVisible := 'False'; ExternalWritable := 'False'} : Word;   // HMI Animation color of the icon
      H_AlarmDWord { ExternalAccessible := 'False'; ExternalVisible := 'False'; ExternalWritable := 'False'} : DWord;   // Alarm Word
   END_VAR
   VAR_IN_OUT
      IO_ETAFuseData : "ETAFuseData";   // ETA fuse status
   END_VAR
   VAR DB_SPECIFIC
      AA_AlarmOFF { ExternalAccessible := 'False'; ExternalVisible := 'False'; ExternalWritable := 'False'} : Bool;   // Fuse Locc-Box is switch OFF / Extra Info ETA Fuse -> Is switch OFF
      AA_AlarmOverload { ExternalAccessible := 'False'; ExternalVisible := 'False'; ExternalWritable := 'False'} : Bool;   // Fuse Locc-Box Blown Alarm / Extra Info ETA Fuse -> Overload Alarm
      AA_AlarmCurrentLimit { ExternalAccessible := 'False'; ExternalVisible := 'False'; ExternalWritable := 'False'} : Bool;   // Fuse Locc-Box Current Limit Alarm / Extra Info ETA Fuse -> Current Limit Alarm
      AA_AlarmUndVolt { ExternalAccessible := 'False'; ExternalVisible := 'False'; ExternalWritable := 'False'} : Bool;   // Fuse Locc-Box Under Voltage Alarm / Extra Info ETA Fuse -> Under Voltage Alarm
      AA_AlarmShortCircuit { ExternalAccessible := 'False'; ExternalVisible := 'False'; ExternalWritable := 'False'} : Bool;   // Fuse Locc-Box Short circuit Alarm / Extra Info ETA Fuse -> Short circuit Alarm
      AA_AlarmTemperature { ExternalAccessible := 'False'; ExternalVisible := 'False'; ExternalWritable := 'False'} : Bool;   // Fuse Locc-Box System error Alarm / Extra Info ETA Fuse -> Temperature Alarm
      AA_FuseName { ExternalAccessible := 'False'; ExternalVisible := 'False'; ExternalWritable := 'False'} : Bool;   // Fuse Locc-Box System error Alarm / Extra Info ETA Fuse -> Fuse name is not found by the config or Instance name DB is wrong OR is found more then one time by the config
      AB_AlarmOFF { ExternalAccessible := 'False'; ExternalVisible := 'False'; ExternalWritable := 'False'} : Bool;   // Fuse Locc-Box is switch OFF / Extra Info ETA Fuse -> Is switch OFF
      AB_AlarmOverload { ExternalAccessible := 'False'; ExternalVisible := 'False'; ExternalWritable := 'False'} : Bool;   // Fuse Locc-Box Blown Alarm / Extra Info ETA Fuse -> Overload Alarm
      AB_AlarmCurrentLimit { ExternalAccessible := 'False'; ExternalVisible := 'False'; ExternalWritable := 'False'} : Bool;   // Fuse Locc-Box Current Limit Alarm / Extra Info ETA Fuse -> Current Limit Alarm
      AB_AlarmUndVolt { ExternalAccessible := 'False'; ExternalVisible := 'False'; ExternalWritable := 'False'} : Bool;   // Fuse Locc-Box Under Voltage Alarm / Extra Info ETA Fuse -> Under Voltage Alarm
      AB_AlarmShortCirc { ExternalAccessible := 'False'; ExternalVisible := 'False'; ExternalWritable := 'False'} : Bool;   // Fuse Locc-Box Short circuit Alarm / Extra Info ETA Fuse -> Short circuit Alarm
      AB_AlarmTemperature { ExternalAccessible := 'False'; ExternalVisible := 'False'; ExternalWritable := 'False'} : Bool;   // Fuse Locc-Box System error Alarm / Extra Info ETA Fuse -> Temperature Alarm
      AB_FuseName { ExternalAccessible := 'False'; ExternalVisible := 'False'; ExternalWritable := 'False'} : Bool;   // Fuse Locc-Box System error Alarm / Extra Info ETA Fuse -> Fuse name is not found by the config or Instance name DB is wrong OR is found more then one time by the config
      AC_AlarmOFF { ExternalAccessible := 'False'; ExternalVisible := 'False'; ExternalWritable := 'False'} : Bool;   // Fuse Locc-Box is switch OFF / Extra Info ETA Fuse -> Is switch OFF
      AC_AlarmOverload { ExternalAccessible := 'False'; ExternalVisible := 'False'; ExternalWritable := 'False'} : Bool;   // Fuse Locc-Box Blown Alarm / Extra Info ETA Fuse -> Overload Alarm
      AC_AlarmCurrentLimit { ExternalAccessible := 'False'; ExternalVisible := 'False'; ExternalWritable := 'False'} : Bool;   // Fuse Locc-Box Current Limit Alarm / Extra Info ETA Fuse -> Current Limit Alarm
      AC_AlarmUndVolt { ExternalAccessible := 'False'; ExternalVisible := 'False'; ExternalWritable := 'False'} : Bool;   // Fuse Locc-Box Under Voltage Alarm / Extra Info ETA Fuse -> Under Voltage Alarm
      AC_AlarmShortCirc { ExternalAccessible := 'False'; ExternalVisible := 'False'; ExternalWritable := 'False'} : Bool;   // Fuse Locc-Box Short circuit Alarm / Extra Info ETA Fuse -> Short circuit Alarm
      AC_AlarmTemperature { ExternalAccessible := 'False'; ExternalVisible := 'False'; ExternalWritable := 'False'} : Bool;   // Fuse Locc-Box System error Alarm / Extra Info ETA Fuse -> Temperature Alarm
      AC_FuseName { ExternalAccessible := 'False'; ExternalVisible := 'False'; ExternalWritable := 'False'} : Bool;   // Fuse Locc-Box System error Alarm / Extra Info ETA Fuse -> Fuse name is not found by the config or Instance name DB is wrong OR is found more then one time by the config
      AD_WarningOFF { ExternalAccessible := 'False'; ExternalVisible := 'False'; ExternalWritable := 'False'} : Bool;   // Fuse Locc-Box OFF Warning / Extra Info ETA Fuse -> OFF Warning
      AD_WarningOverload { ExternalAccessible := 'False'; ExternalVisible := 'False'; ExternalWritable := 'False'} : Bool;   // Fuse Locc-Box Blown Warning / Extra Info ETA Fuse -> Overload Warning
      AD_WarningCurrentLimit { ExternalAccessible := 'False'; ExternalVisible := 'False'; ExternalWritable := 'False'} : Bool;   // Fuse Locc-Box Current Limit Warning / Extra Info ETA Fuse -> Current Limit Warning
      AD_WarningUndVolt { ExternalAccessible := 'False'; ExternalVisible := 'False'; ExternalWritable := 'False'} : Bool;   // Fuse Locc-Box Under Voltage Warning / Extra Info ETA Fuse -> Under Voltage Warning
      AD_WarningShortCirc { ExternalAccessible := 'False'; ExternalVisible := 'False'; ExternalWritable := 'False'} : Bool;   // Fuse Locc-Box Short circuit Warning / Extra Info ETA Fuse -> Short circuit Warning
      AD_WarningTemperature { ExternalAccessible := 'False'; ExternalVisible := 'False'; ExternalWritable := 'False'} : Bool;   // Fuse Locc-Box System error Warning / Extra Info ETA Fuse -> Temperature Warning
      AD_WarningFuseName { ExternalAccessible := 'False'; ExternalVisible := 'False'; ExternalWritable := 'False'} : Bool;   // Fuse Locc-Box System error Alarm / Extra Info ETA Fuse -> Fuse name is not found by the config or Instance name DB is wrong OR is found more then one time by the config
      AD_NominalCurrent { ExternalAccessible := 'False'; ExternalVisible := 'False'; ExternalWritable := 'False'} : Bool;   // Rotary switch on the fuse is changed for the current / Extra Info ETA Fuse -> Nominal Current for the fuse is changed
      H_HMICmd : Word;   // HMI Command from Pop-Up
      H_Out : Struct   // HMI
         Anim : Word;   // HMI Animation Word
         Anim2 : Word;   // HMI Animation Word
         Anim3 : Word;   // HMI Animation Word
         Voltage : Real;   // HMI Input Voltage / HMI Voltage
         Current : Real;   // HMI Input Voltage / HMI Current
         NominalCurrent : Int;   // HMI Current setpoint / HMI Nominal Current
         NominalCurrentConfig : Int;   // HMI Current setpoint / HMI Nominal Current Config
         "Name" : String[40];   // HMI Name
         Description : String[60];   // HMI Description
         DBnr : Int;   // HMI Animation DB number
      END_STRUCT;
      FuseNr { ExternalAccessible := 'False'; ExternalVisible := 'False'; ExternalWritable := 'False'} : Int;   // Fuse number in struct "ETAFuseStatus"
      AlarmOFF { ExternalAccessible := 'False'; ExternalVisible := 'False'; ExternalWritable := 'False'} : Bool;   // Fuse Locc-Box is switch OFF / Fuse ETA Is switch OFF
      AlarmOverload { ExternalAccessible := 'False'; ExternalVisible := 'False'; ExternalWritable := 'False'} : Bool;   // Fuse Locc-Box Blown Alarm / Fuse ETA Overload Alarm
      AlarmCurrentLimit { ExternalAccessible := 'False'; ExternalVisible := 'False'; ExternalWritable := 'False'} : Bool;   // Fuse Locc-Box Current Limit Alarm / Fuse ETA Current Limit Alarm
      AlarmUndVolt { ExternalAccessible := 'False'; ExternalVisible := 'False'; ExternalWritable := 'False'} : Bool;   // Fuse Locc-Box Under Voltage Alarm / Fuse ETA Under Voltage Alarm
      AlarmShortCirc { ExternalAccessible := 'False'; ExternalVisible := 'False'; ExternalWritable := 'False'} : Bool;   // Fuse Locc-Box Short circuit Alarm / Fuse ETA Short circuit Alarm
      AlarmTemperature { ExternalAccessible := 'False'; ExternalVisible := 'False'; ExternalWritable := 'False'} : Bool;   // Fuse Locc-Box System error Alarm / Fuse ETA Temperature Alarm
      AlarmFuseName { ExternalAccessible := 'False'; ExternalVisible := 'False'; ExternalWritable := 'False'} : Bool;   // Fuse Locc-Box System error Alarm / Fuse ETA Fuse Name Alarm
      AlarmCondOFF { ExternalAccessible := 'False'; ExternalVisible := 'False'; ExternalWritable := 'False'} : Bool;   // Alarm condition
      AlarmCondOverload { ExternalAccessible := 'False'; ExternalVisible := 'False'; ExternalWritable := 'False'} : Bool;   // Alarm condition
      AlarmCondCurrentLimit { ExternalAccessible := 'False'; ExternalVisible := 'False'; ExternalWritable := 'False'} : Bool;   // Alarm condition
      AlarmCondUndVolt { ExternalAccessible := 'False'; ExternalVisible := 'False'; ExternalWritable := 'False'} : Bool;   // Alarm condition
      AlarmCondShortCirc { ExternalAccessible := 'False'; ExternalVisible := 'False'; ExternalWritable := 'False'} : Bool;   // Alarm condition
      AlarmCondTemperature { ExternalAccessible := 'False'; ExternalVisible := 'False'; ExternalWritable := 'False'} : Bool;   // Alarm condition
      AlarmCondFuseName { ExternalAccessible := 'False'; ExternalVisible := 'False'; ExternalWritable := 'False'} : Bool;   // Alarm condition
      Alarm { ExternalAccessible := 'False'; ExternalVisible := 'False'; ExternalWritable := 'False'} : Bool;   // Alarm
      Warning { ExternalAccessible := 'False'; ExternalVisible := 'False'; ExternalWritable := 'False'} : Bool;   // Warning
      AlarmClass_A { ExternalAccessible := 'False'; ExternalVisible := 'False'; ExternalWritable := 'False'} : Bool;   // The alarm is from alarm class A
      AlarmClass_B { ExternalAccessible := 'False'; ExternalVisible := 'False'; ExternalWritable := 'False'} : Bool;   // The alarm is from alarm class B
      AlarmClass_C { ExternalAccessible := 'False'; ExternalVisible := 'False'; ExternalWritable := 'False'} : Bool;   // The alarm is from alarm class C
      AlarmClass_D { ExternalAccessible := 'False'; ExternalVisible := 'False'; ExternalWritable := 'False'} : Bool;   // The alarm is from alarm class C / The alarm is from alarm class D
      C_LevelOFF { ExternalAccessible := 'False'; ExternalVisible := 'False'; ExternalWritable := 'False'} : Bool;   // Config alarm level
      C_LevelOverload { ExternalAccessible := 'False'; ExternalVisible := 'False'; ExternalWritable := 'False'} : Bool;   // Config alarm level
      C_LevelCurrentLimit { ExternalAccessible := 'False'; ExternalVisible := 'False'; ExternalWritable := 'False'} : Bool;   // Config alarm level
      C_LevelUndVolt { ExternalAccessible := 'False'; ExternalVisible := 'False'; ExternalWritable := 'False'} : Bool;   // Config alarm level
      C_LevelShortCirc { ExternalAccessible := 'False'; ExternalVisible := 'False'; ExternalWritable := 'False'} : Bool;   // Config alarm level
      C_LevelTemperature { ExternalAccessible := 'False'; ExternalVisible := 'False'; ExternalWritable := 'False'} : Bool;   // Config alarm level
      C_LevelFuseName { ExternalAccessible := 'False'; ExternalVisible := 'False'; ExternalWritable := 'False'} : Bool;   // Config alarm level
      C_LevelSpareBit7 { ExternalAccessible := 'False'; ExternalVisible := 'False'; ExternalWritable := 'False'} : Bool;   // Config alarm level
      C_LevelSpareBit8 { ExternalAccessible := 'False'; ExternalVisible := 'False'; ExternalWritable := 'False'} : Bool;   // Config alarm level
      C_LevelSpareBit9 { ExternalAccessible := 'False'; ExternalVisible := 'False'; ExternalWritable := 'False'} : Bool;   // Config alarm level
      C_LevelSpareBit10 { ExternalAccessible := 'False'; ExternalVisible := 'False'; ExternalWritable := 'False'} : Bool;   // Config alarm level
      C_LevelSpareBit11 { ExternalAccessible := 'False'; ExternalVisible := 'False'; ExternalWritable := 'False'} : Bool;   // Config alarm level
      C_LevelSpareBit12 { ExternalAccessible := 'False'; ExternalVisible := 'False'; ExternalWritable := 'False'} : Bool;   // Config alarm level
      C_LevelSpareBit13 { ExternalAccessible := 'False'; ExternalVisible := 'False'; ExternalWritable := 'False'} : Bool;   // Config alarm level
      C_LevelSpareBit14 { ExternalAccessible := 'False'; ExternalVisible := 'False'; ExternalWritable := 'False'} : Bool;   // Config alarm level
      C_LevelSpareBit15 { ExternalAccessible := 'False'; ExternalVisible := 'False'; ExternalWritable := 'False'} : Bool;   // Config alarm level
      HMICmdSwitchON { ExternalAccessible := 'False'; ExternalVisible := 'False'; ExternalWritable := 'False'} : Bool;   // HMICmd
      HMICmdSwitchOFF { ExternalAccessible := 'False'; ExternalVisible := 'False'; ExternalWritable := 'False'} : Bool;   // HMICmd
      HMICmdResetOFF { ExternalAccessible := 'False'; ExternalVisible := 'False'; ExternalWritable := 'False'} : Bool;   // HMICmd
      HMICmdResetOverload { ExternalAccessible := 'False'; ExternalVisible := 'False'; ExternalWritable := 'False'} : Bool;   // HMICmd
      HMICmdSpareBit2 { ExternalAccessible := 'False'; ExternalVisible := 'False'; ExternalWritable := 'False'} : Bool;   // HMICmd
      HMICmdResetCurrentLimit { ExternalAccessible := 'False'; ExternalVisible := 'False'; ExternalWritable := 'False'} : Bool;   // HMICmd
      HMICmdResetUndVolt { ExternalAccessible := 'False'; ExternalVisible := 'False'; ExternalWritable := 'False'} : Bool;   // HMICmd
      HMICmdResetShortCirc { ExternalAccessible := 'False'; ExternalVisible := 'False'; ExternalWritable := 'False'} : Bool;   // HMICmd
      HMICmdResetTemperature { ExternalAccessible := 'False'; ExternalVisible := 'False'; ExternalWritable := 'False'} : Bool;   // HMICmd
      HMICmdTrsf { ExternalAccessible := 'False'; ExternalVisible := 'False'; ExternalWritable := 'False'} : Bool;   // HMICmd
      HMICmdReset { ExternalAccessible := 'False'; ExternalVisible := 'False'; ExternalWritable := 'False'} : Bool;   // HMICmd
      HMICmdSpareBit11 { ExternalAccessible := 'False'; ExternalVisible := 'False'; ExternalWritable := 'False'} : Bool;   // HMICmd
      HMICmdSpareBit12 { ExternalAccessible := 'False'; ExternalVisible := 'False'; ExternalWritable := 'False'} : Bool;   // HMICmd
      HMICmdSpareBit13 { ExternalAccessible := 'False'; ExternalVisible := 'False'; ExternalWritable := 'False'} : Bool;   // HMICmd
      HMICmdSpareBit14 { ExternalAccessible := 'False'; ExternalVisible := 'False'; ExternalWritable := 'False'} : Bool;   // HMICmd
      HMICmdSpareBit15 { ExternalAccessible := 'False'; ExternalVisible := 'False'; ExternalWritable := 'False'} : Bool;   // HMICmd
      C_LocalResetOFF { ExternalAccessible := 'False'; ExternalVisible := 'False'; ExternalWritable := 'False'} : Bool;   // Config Local reset
      C_LocalResetOverload { ExternalAccessible := 'False'; ExternalVisible := 'False'; ExternalWritable := 'False'} : Bool;   // Config Local reset
      C_LocalResetCurrentLimit { ExternalAccessible := 'False'; ExternalVisible := 'False'; ExternalWritable := 'False'} : Bool;   // Config Local reset
      C_LocalResetUndVolt { ExternalAccessible := 'False'; ExternalVisible := 'False'; ExternalWritable := 'False'} : Bool;   // Config Local reset
      C_LocalResetShortCirc { ExternalAccessible := 'False'; ExternalVisible := 'False'; ExternalWritable := 'False'} : Bool;   // Config Local reset
      C_LocalResetTemperature { ExternalAccessible := 'False'; ExternalVisible := 'False'; ExternalWritable := 'False'} : Bool;   // Config Local reset
      C_LocalResetSpareBit6 { ExternalAccessible := 'False'; ExternalVisible := 'False'; ExternalWritable := 'False'} : Bool;   // Config Local reset
      C_LocalResetSpareBit7 { ExternalAccessible := 'False'; ExternalVisible := 'False'; ExternalWritable := 'False'} : Bool;   // Config Local reset
      C_LocalResetSpareBit8 { ExternalAccessible := 'False'; ExternalVisible := 'False'; ExternalWritable := 'False'} : Bool;   // Config Local reset
      C_LocalResetSpareBit9 { ExternalAccessible := 'False'; ExternalVisible := 'False'; ExternalWritable := 'False'} : Bool;   // Config Local reset
      C_LocalResetSpareBit10 { ExternalAccessible := 'False'; ExternalVisible := 'False'; ExternalWritable := 'False'} : Bool;   // Config Local reset
      C_LocalResetSpareBit11 { ExternalAccessible := 'False'; ExternalVisible := 'False'; ExternalWritable := 'False'} : Bool;   // Config Local reset
      C_LocalResetSpareBit12 { ExternalAccessible := 'False'; ExternalVisible := 'False'; ExternalWritable := 'False'} : Bool;   // Config Local reset
      C_LocalResetSpareBit13 { ExternalAccessible := 'False'; ExternalVisible := 'False'; ExternalWritable := 'False'} : Bool;   // Config Local reset
      C_LocalResetSpareBit14 { ExternalAccessible := 'False'; ExternalVisible := 'False'; ExternalWritable := 'False'} : Bool;   // Config Local reset
      C_LocalResetSpareBit15 { ExternalAccessible := 'False'; ExternalVisible := 'False'; ExternalWritable := 'False'} : Bool;   // Config Local reset
      DBnr { ExternalAccessible := 'False'; ExternalVisible := 'False'; ExternalWritable := 'False'} : Int;   // DB number / HMI DB number
      DBName { ExternalAccessible := 'False'; ExternalVisible := 'False'; ExternalWritable := 'False'} : String[40];   // DB Name
      FuseNameOK { ExternalAccessible := 'False'; ExternalVisible := 'False'; ExternalWritable := 'False'} : Bool;   // Fuse name is found one time by the config
      FuseNameNOK { ExternalAccessible := 'False'; ExternalVisible := 'False'; ExternalWritable := 'False'} : Bool;   // Fuse name is not found by the config or Instance name DB is wrong
      FuseNameMoreThenOne { ExternalAccessible := 'False'; ExternalVisible := 'False'; ExternalWritable := 'False'} : Bool;   // Fuse name is found more then one time by the config
      StatusNotAvailable { ExternalAccessible := 'False'; ExternalVisible := 'False'; ExternalWritable := 'False'} : Bool;   // Status not available
      Edge { ExternalAccessible := 'False'; ExternalVisible := 'False'; ExternalWritable := 'False'} : Bool;   // Flank
      Status { ExternalAccessible := 'False'; ExternalVisible := 'False'; ExternalWritable := 'False'} : Struct   // Status Fuse
         LoadOutput { ExternalAccessible := 'False'; ExternalVisible := 'False'; ExternalWritable := 'False'} : Bool;   // Load Output
         ShortCircuit { ExternalAccessible := 'False'; ExternalVisible := 'False'; ExternalWritable := 'False'} : Bool;   // Short Circuit
         Overload { ExternalAccessible := 'False'; ExternalVisible := 'False'; ExternalWritable := 'False'} : Bool;   // Overload
         LowVoltage { ExternalAccessible := 'False'; ExternalVisible := 'False'; ExternalWritable := 'False'} : Bool;   // Low Voltage
         ExcessTemparature1 { ExternalAccessible := 'False'; ExternalVisible := 'False'; ExternalWritable := 'False'} : Bool;   // Excess Temparature1
         ExcessTemparature2 { ExternalAccessible := 'False'; ExternalVisible := 'False'; ExternalWritable := 'False'} : Bool;   // Excess Temparature2
         LimitValueCurrent { ExternalAccessible := 'False'; ExternalVisible := 'False'; ExternalWritable := 'False'} : Bool;   // Limit Value Current
         Event { ExternalAccessible := 'False'; ExternalVisible := 'False'; ExternalWritable := 'False'} : Bool;   // Event
      END_STRUCT;
      T_ResetControl { ExternalAccessible := 'False'; ExternalVisible := 'False'; ExternalWritable := 'False'} : TON_TIME;   // Timer
   END_VAR
   VAR_TEMP
      TmpWString : WString;
   END_VAR
   VAR_TEMP   // added for the SCL form of the ladder/FBD networks
      _w1 : Bool;
   END_VAR
BEGIN

NETWORK
TITLE = **** 1 - Inputs **** DB number
// DB number
      L     DINO;
      T     #DBnr;

REGION Network 2: **** 1 - Inputs **** DB name
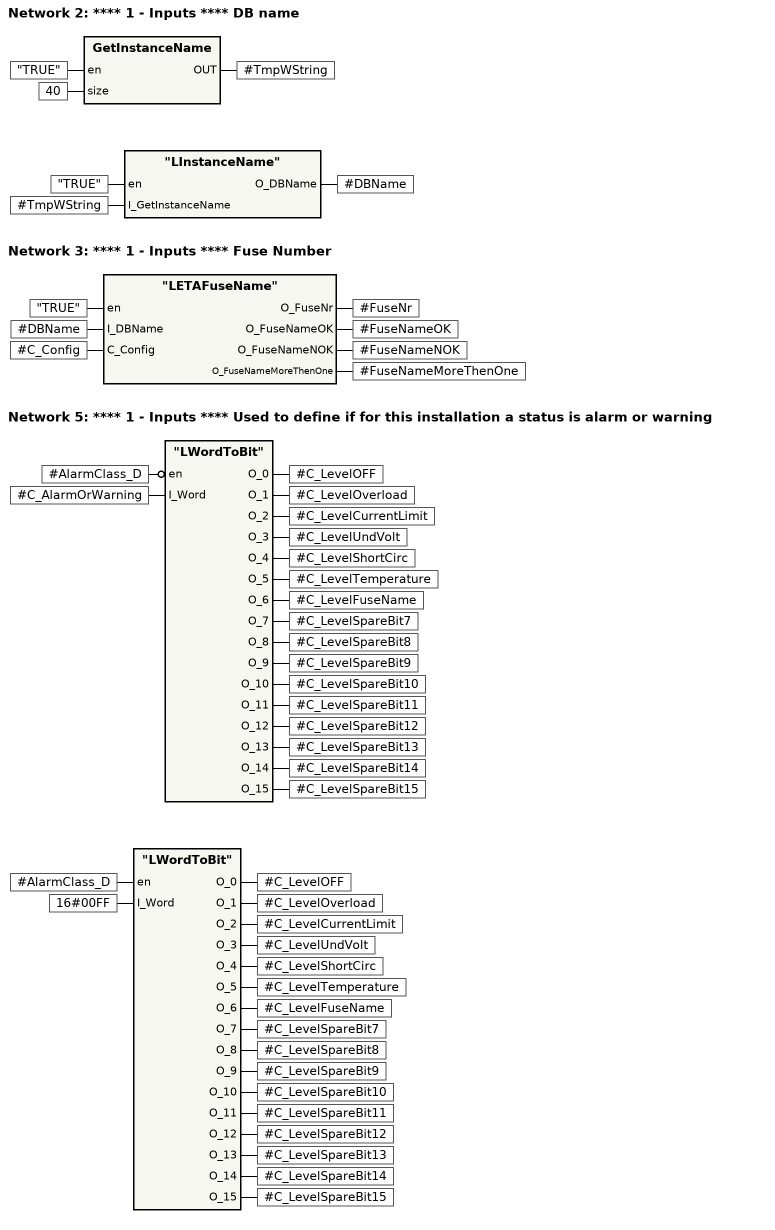
   IF "TRUE" THEN GetInstanceName(size := 40, OUT => #TmpWString); END_IF;
   IF "TRUE" THEN "LInstanceName"(I_GetInstanceName := #TmpWString, O_DBName => #DBName); END_IF;
END_REGION

REGION Network 3: **** 1 - Inputs **** Fuse Number
   IF "TRUE" THEN
       "LETAFuseName"(I_DBName := #DBName,
                      C_Config := #C_Config,
                      O_FuseNr => #FuseNr,
                      O_FuseNameOK => #FuseNameOK,
                      O_FuseNameNOK => #FuseNameNOK,
                      O_FuseNameMoreThenOne => #FuseNameMoreThenOne);
   END_IF;
END_REGION

NETWORK
TITLE = **** 1 - Inputs **** Alarm class
// Alarm class
// Alarm class = D
      L     #I_AlarmClass;
      L     'D';
      ==I;
      =     #AlarmClass_D;

// Alarm class = C
      L     #I_AlarmClass;
      L     'C';
      ==I;
      =     #AlarmClass_C;

// Alarm class = B
      L     #I_AlarmClass;
      L     'B';
      ==I;
      =     #AlarmClass_B;

// Alarm class = A
      AN    #AlarmClass_B;
      AN    #AlarmClass_C;
      AN    #AlarmClass_D;
      =     #AlarmClass_A;


REGION Network 5: **** 1 - Inputs **** Used to define if for this installation a status is alarm or warning
   // Extract the configuration
   // Used to define if for this installation a status is alarm or warning
   IF NOT #AlarmClass_D THEN
       "LWordToBit"(I_Word := #C_AlarmOrWarning,
                    O_0 => #C_LevelOFF,
                    O_1 => #C_LevelOverload,
                    O_2 => #C_LevelCurrentLimit,
                    O_3 => #C_LevelUndVolt,
                    O_4 => #C_LevelShortCirc,
                    O_5 => #C_LevelTemperature,
                    O_6 => #C_LevelFuseName,
                    O_7 => #C_LevelSpareBit7,
                    O_8 => #C_LevelSpareBit8,
                    O_9 => #C_LevelSpareBit9,
                    O_10 => #C_LevelSpareBit10,
                    O_11 => #C_LevelSpareBit11,
                    O_12 => #C_LevelSpareBit12,
                    O_13 => #C_LevelSpareBit13,
                    O_14 => #C_LevelSpareBit14,
                    O_15 => #C_LevelSpareBit15);
   END_IF;
   IF #AlarmClass_D THEN
       "LWordToBit"(I_Word := 16#00FF,
                    O_0 => #C_LevelOFF,
                    O_1 => #C_LevelOverload,
                    O_2 => #C_LevelCurrentLimit,
                    O_3 => #C_LevelUndVolt,
                    O_4 => #C_LevelShortCirc,
                    O_5 => #C_LevelTemperature,
                    O_6 => #C_LevelFuseName,
                    O_7 => #C_LevelSpareBit7,
                    O_8 => #C_LevelSpareBit8,
                    O_9 => #C_LevelSpareBit9,
                    O_10 => #C_LevelSpareBit10,
                    O_11 => #C_LevelSpareBit11,
                    O_12 => #C_LevelSpareBit12,
                    O_13 => #C_LevelSpareBit13,
                    O_14 => #C_LevelSpareBit14,
                    O_15 => #C_LevelSpareBit15);
   END_IF;
END_REGION

REGION Network 6: **** 1 - Inputs **** Used to define if for this installation an error is local or remote reset
   // Extract the configuration
   // Used to define if for this installation an error is local or remote reset
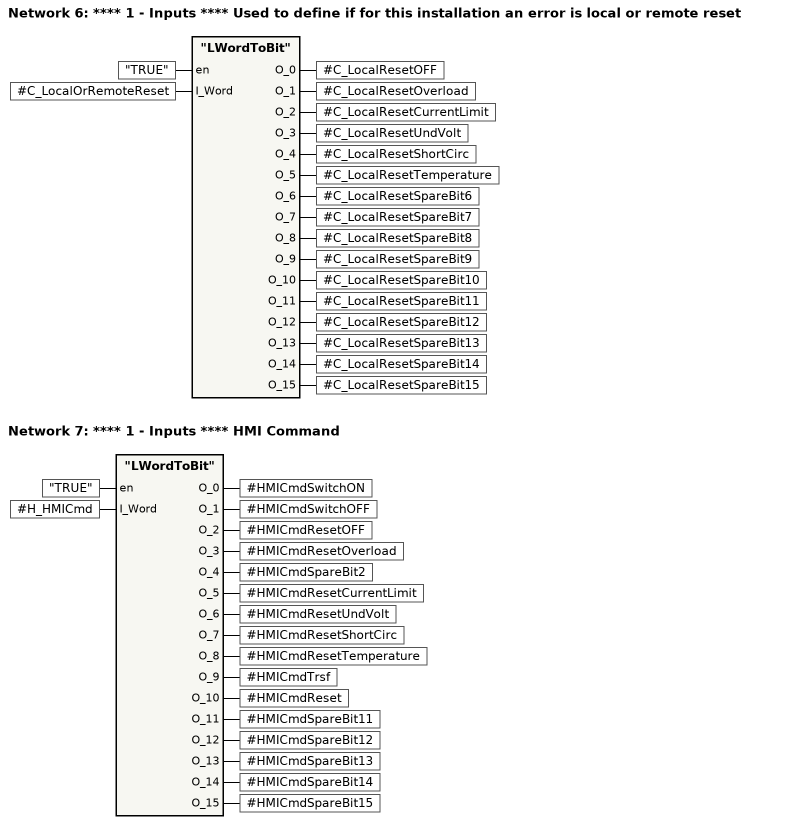
   IF "TRUE" THEN
       "LWordToBit"(I_Word := #C_LocalOrRemoteReset,
                    O_0 => #C_LocalResetOFF,
                    O_1 => #C_LocalResetOverload,
                    O_2 => #C_LocalResetCurrentLimit,
                    O_3 => #C_LocalResetUndVolt,
                    O_4 => #C_LocalResetShortCirc,
                    O_5 => #C_LocalResetTemperature,
                    O_6 => #C_LocalResetSpareBit6,
                    O_7 => #C_LocalResetSpareBit7,
                    O_8 => #C_LocalResetSpareBit8,
                    O_9 => #C_LocalResetSpareBit9,
                    O_10 => #C_LocalResetSpareBit10,
                    O_11 => #C_LocalResetSpareBit11,
                    O_12 => #C_LocalResetSpareBit12,
                    O_13 => #C_LocalResetSpareBit13,
                    O_14 => #C_LocalResetSpareBit14,
                    O_15 => #C_LocalResetSpareBit15);
   END_IF;
END_REGION

REGION Network 7: **** 1 - Inputs **** HMI Command
   // Extract the HMI command bit
   // Command bit from HMI
   IF "TRUE" THEN
       "LWordToBit"(I_Word := #H_HMICmd,
                    O_0 => #HMICmdSwitchON,
                    O_1 => #HMICmdSwitchOFF,
                    O_2 => #HMICmdResetOFF,
                    O_3 => #HMICmdResetOverload,
                    O_4 => #HMICmdSpareBit2,
                    O_5 => #HMICmdResetCurrentLimit,
                    O_6 => #HMICmdResetUndVolt,
                    O_7 => #HMICmdResetShortCirc,
                    O_8 => #HMICmdResetTemperature,
                    O_9 => #HMICmdTrsf,
                    O_10 => #HMICmdReset,
                    O_11 => #HMICmdSpareBit11,
                    O_12 => #HMICmdSpareBit12,
                    O_13 => #HMICmdSpareBit13,
                    O_14 => #HMICmdSpareBit14,
                    O_15 => #HMICmdSpareBit15);
   END_IF;
END_REGION

REGION Network 8: **** 1 - Inputs **** Status
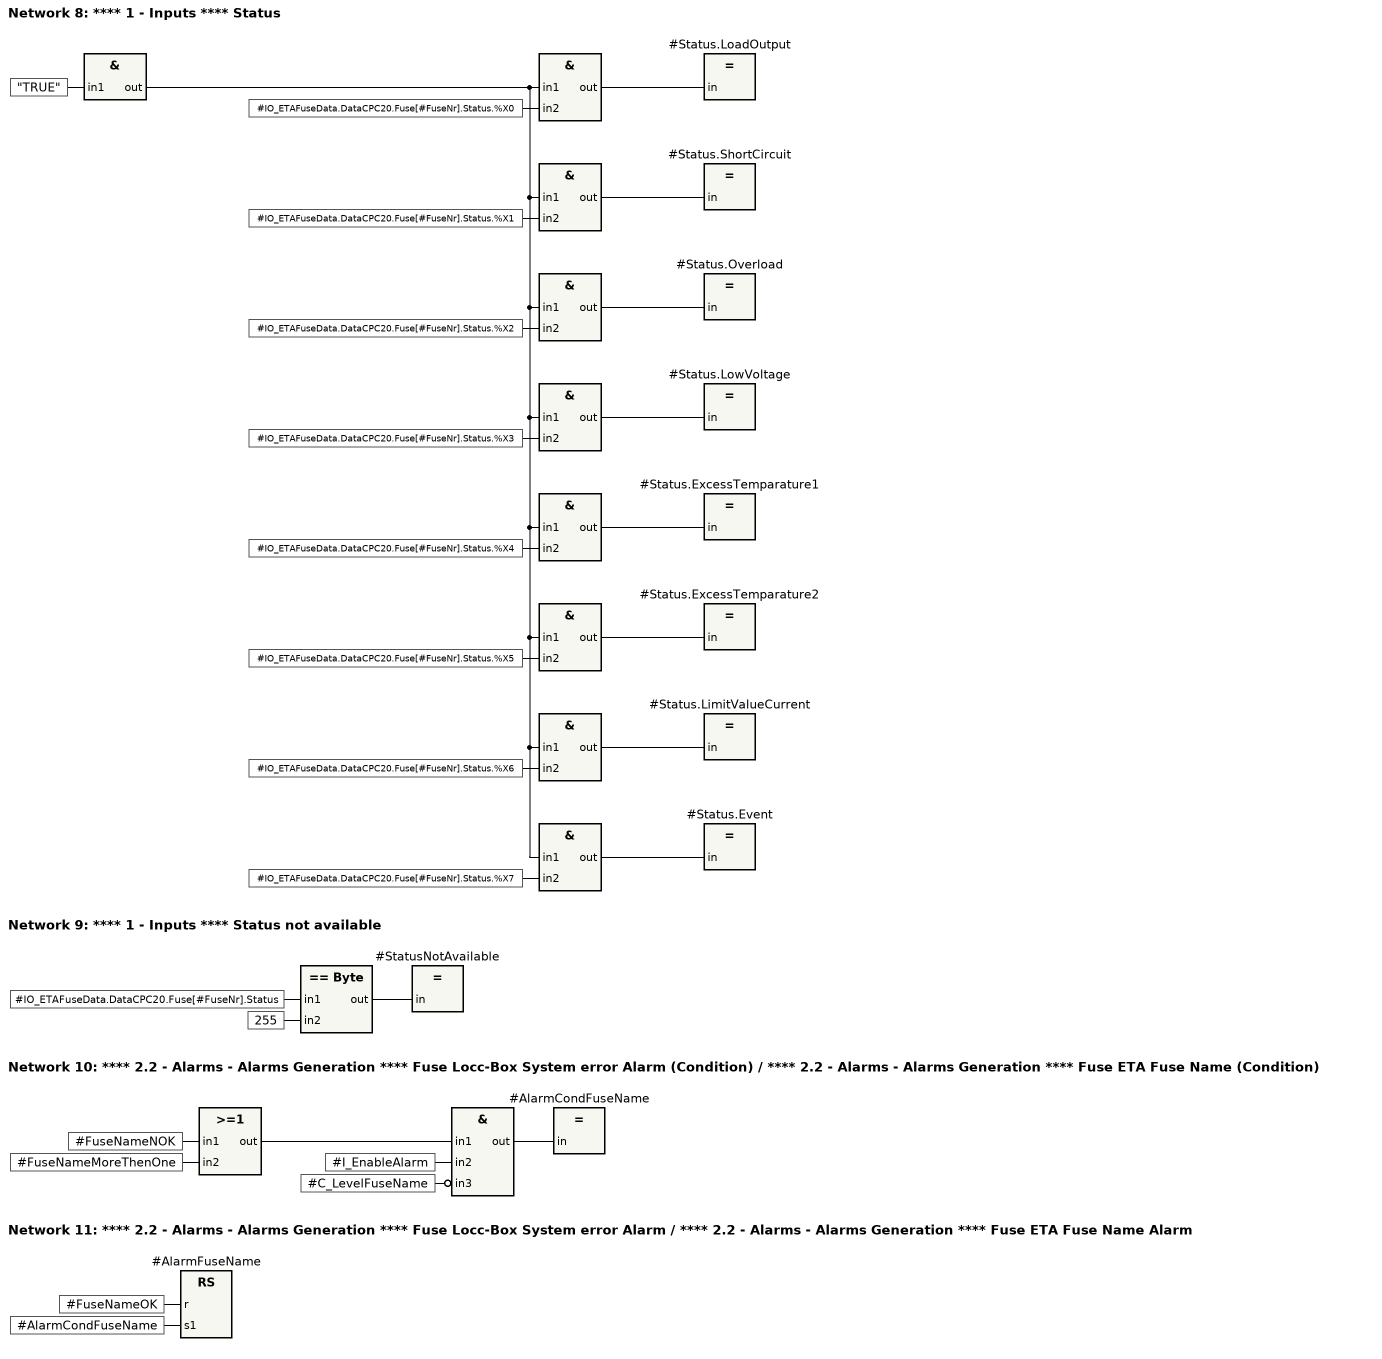
   #Status.LoadOutput := "TRUE" AND #IO_ETAFuseData.DataCPC20.Fuse[#FuseNr].Status.%X0;
   #Status.ShortCircuit := "TRUE" AND #IO_ETAFuseData.DataCPC20.Fuse[#FuseNr].Status.%X1;
   #Status.Overload := "TRUE" AND #IO_ETAFuseData.DataCPC20.Fuse[#FuseNr].Status.%X2;
   #Status.LowVoltage := "TRUE" AND #IO_ETAFuseData.DataCPC20.Fuse[#FuseNr].Status.%X3;
   #Status.ExcessTemparature1 := "TRUE" AND #IO_ETAFuseData.DataCPC20.Fuse[#FuseNr].Status.%X4;
   #Status.ExcessTemparature2 := "TRUE" AND #IO_ETAFuseData.DataCPC20.Fuse[#FuseNr].Status.%X5;
   #Status.LimitValueCurrent := "TRUE" AND #IO_ETAFuseData.DataCPC20.Fuse[#FuseNr].Status.%X6;
   #Status.Event := "TRUE" AND #IO_ETAFuseData.DataCPC20.Fuse[#FuseNr].Status.%X7;
END_REGION

REGION Network 9: **** 1 - Inputs **** Status not available
   #StatusNotAvailable := #IO_ETAFuseData.DataCPC20.Fuse[#FuseNr].Status = 255;
END_REGION

REGION Network 10: **** 2.2 - Alarms - Alarms Generation **** Fuse Locc-Box System error Alarm (Condition) / **** 2.2 - Alarms - Alarms Generation **** Fuse ETA Fuse Name (Condition)
   // Condition for the Alarm
   #AlarmCondFuseName := (#FuseNameNOK OR #FuseNameMoreThenOne) AND #I_EnableAlarm AND NOT #C_LevelFuseName;
END_REGION

REGION Network 11: **** 2.2 - Alarms - Alarms Generation **** Fuse Locc-Box System error Alarm / **** 2.2 - Alarms - Alarms Generation **** Fuse ETA Fuse Name Alarm
   // Memorisation of the Alarm
   IF #FuseNameOK THEN
       #AlarmFuseName := FALSE;   // RS flip-flop
   END_IF;
   IF #AlarmCondFuseName THEN #AlarmFuseName := TRUE; END_IF;
END_REGION

REGION Network 12: **** 2.2 - Alarms - Alarms Generation **** Fuse Locc-Box System error Warning / **** 2.2 - Alarms - Alarms Generation **** Fuse ETA Fuse Name Warning
   // Memorisation of the Alarm
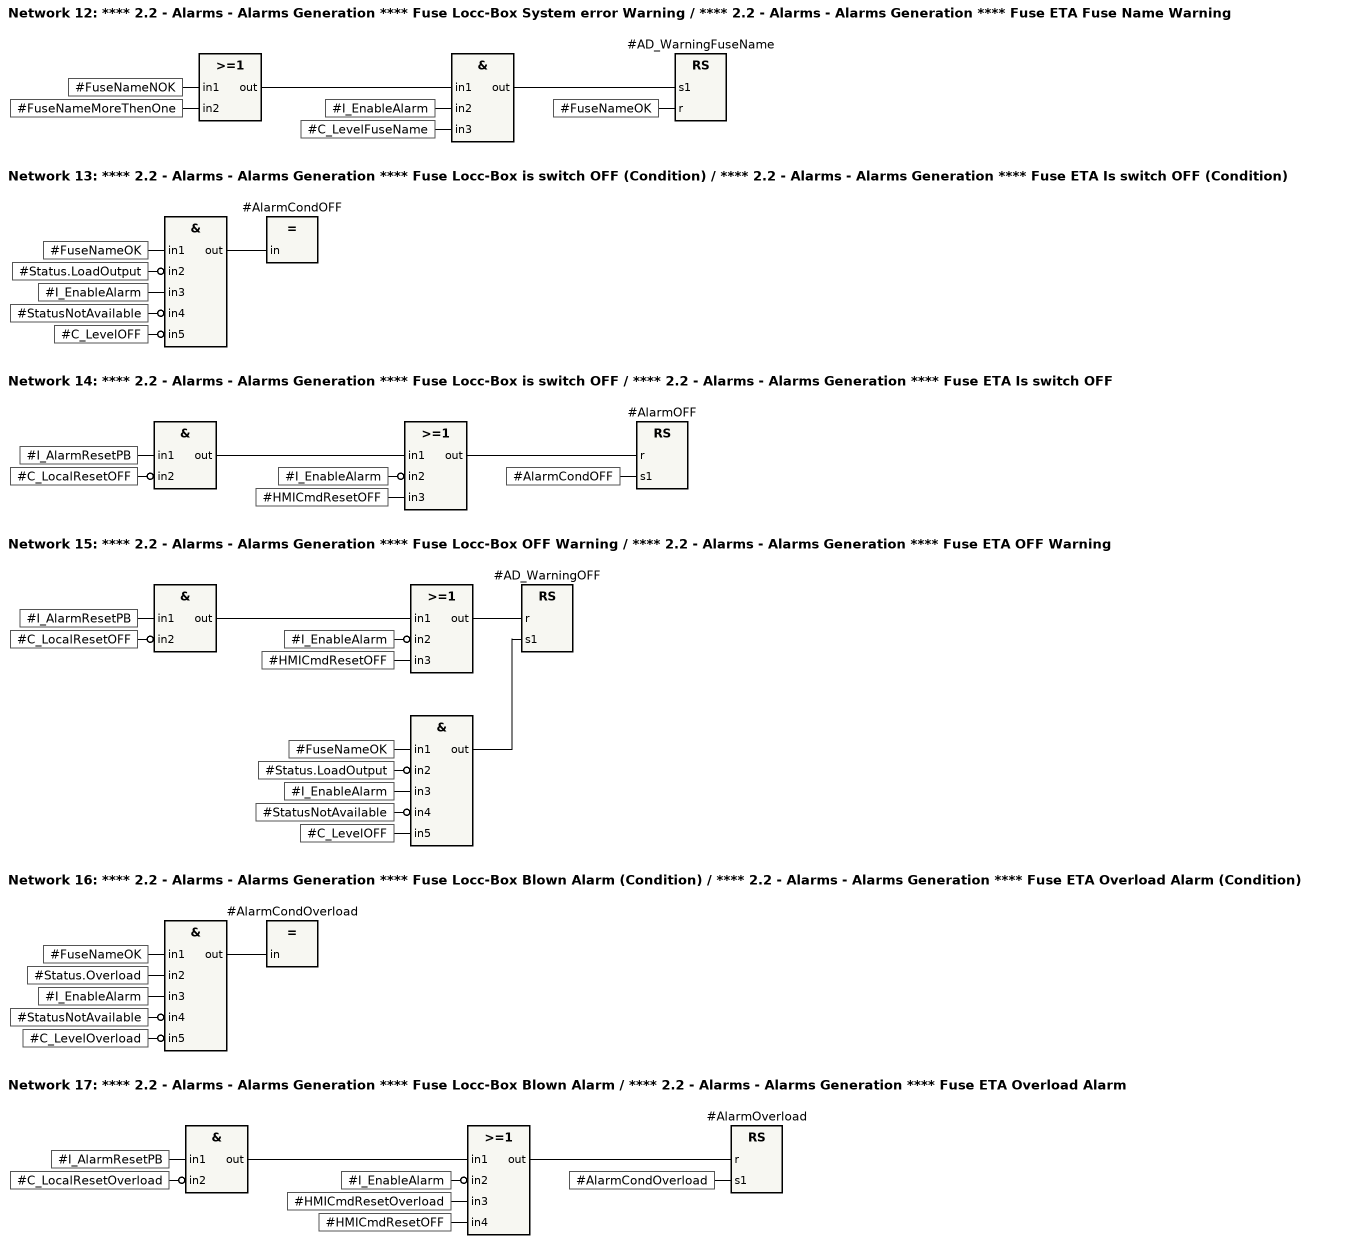
   IF #FuseNameOK THEN
       #AD_WarningFuseName := FALSE;   // RS flip-flop
   END_IF;
   IF (#FuseNameNOK OR #FuseNameMoreThenOne) AND #I_EnableAlarm AND #C_LevelFuseName THEN
       #AD_WarningFuseName := TRUE;
   END_IF;
END_REGION

REGION Network 13: **** 2.2 - Alarms - Alarms Generation **** Fuse Locc-Box is switch OFF (Condition) / **** 2.2 - Alarms - Alarms Generation **** Fuse ETA Is switch OFF (Condition)
   // Condition for the Alarm
   #AlarmCondOFF := #FuseNameOK AND NOT #Status.LoadOutput AND #I_EnableAlarm AND NOT #StatusNotAvailable AND NOT #C_LevelOFF;
END_REGION

REGION Network 14: **** 2.2 - Alarms - Alarms Generation **** Fuse Locc-Box is switch OFF / **** 2.2 - Alarms - Alarms Generation **** Fuse ETA Is switch OFF
   // Memorisation of the Alarm
   IF (#I_AlarmResetPB AND NOT #C_LocalResetOFF) OR NOT #I_EnableAlarm OR #HMICmdResetOFF THEN
       #AlarmOFF := FALSE;   // RS flip-flop
   END_IF;
   IF #AlarmCondOFF THEN #AlarmOFF := TRUE; END_IF;
END_REGION

REGION Network 15: **** 2.2 - Alarms - Alarms Generation **** Fuse Locc-Box OFF Warning / **** 2.2 - Alarms - Alarms Generation **** Fuse ETA OFF Warning
   // Memorisation of the Alarm
   IF (#I_AlarmResetPB AND NOT #C_LocalResetOFF) OR NOT #I_EnableAlarm OR #HMICmdResetOFF THEN
       #AD_WarningOFF := FALSE;   // RS flip-flop
   END_IF;
   IF #FuseNameOK AND NOT #Status.LoadOutput AND #I_EnableAlarm AND NOT #StatusNotAvailable AND #C_LevelOFF THEN
       #AD_WarningOFF := TRUE;
   END_IF;
END_REGION

REGION Network 16: **** 2.2 - Alarms - Alarms Generation **** Fuse Locc-Box Blown Alarm (Condition) / **** 2.2 - Alarms - Alarms Generation **** Fuse ETA Overload Alarm (Condition)
   // Condition for the Alarm
   #AlarmCondOverload := #FuseNameOK AND #Status.Overload AND #I_EnableAlarm AND NOT #StatusNotAvailable AND NOT #C_LevelOverload;
END_REGION

REGION Network 17: **** 2.2 - Alarms - Alarms Generation **** Fuse Locc-Box Blown Alarm / **** 2.2 - Alarms - Alarms Generation **** Fuse ETA Overload Alarm
   // Memorisation of the Alarm
   IF (#I_AlarmResetPB AND NOT #C_LocalResetOverload) OR NOT #I_EnableAlarm OR #HMICmdResetOverload OR #HMICmdResetOFF THEN
       #AlarmOverload := FALSE;   // RS flip-flop
   END_IF;
   IF #AlarmCondOverload THEN #AlarmOverload := TRUE; END_IF;
END_REGION

REGION Network 18: **** 2.2 - Alarms - Alarms Generation **** Fuse Locc-Box Blown Warning / **** 2.2 - Alarms - Alarms Generation **** Fuse ETA Overload Warning
   // Memorisation of the Alarm
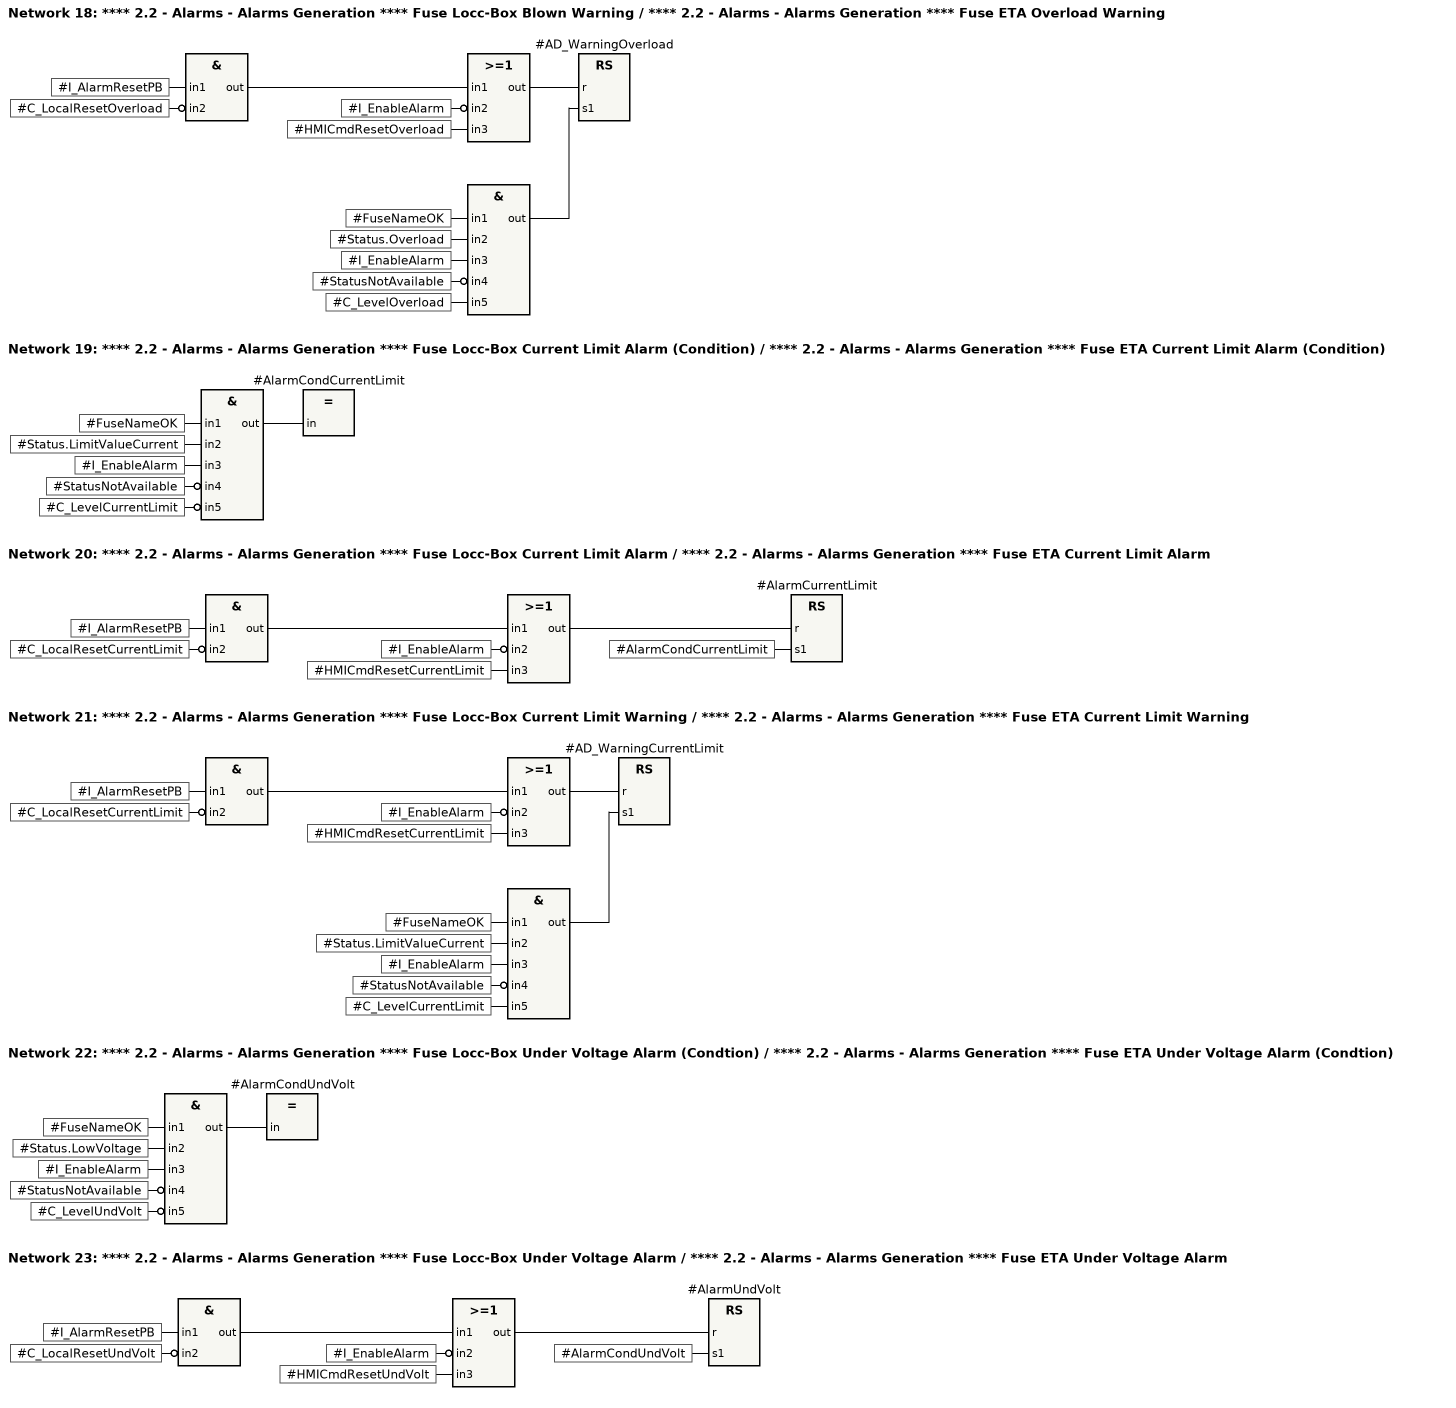
   IF (#I_AlarmResetPB AND NOT #C_LocalResetOverload) OR NOT #I_EnableAlarm OR #HMICmdResetOverload THEN
       #AD_WarningOverload := FALSE;   // RS flip-flop
   END_IF;
   IF #FuseNameOK AND #Status.Overload AND #I_EnableAlarm AND NOT #StatusNotAvailable AND #C_LevelOverload THEN
       #AD_WarningOverload := TRUE;
   END_IF;
END_REGION

REGION Network 19: **** 2.2 - Alarms - Alarms Generation **** Fuse Locc-Box Current Limit Alarm (Condition) / **** 2.2 - Alarms - Alarms Generation **** Fuse ETA Current Limit Alarm (Condition)
   // Condition for the Alarm
   #AlarmCondCurrentLimit := #FuseNameOK AND #Status.LimitValueCurrent AND #I_EnableAlarm AND NOT #StatusNotAvailable AND NOT #C_LevelCurrentLimit;
END_REGION

REGION Network 20: **** 2.2 - Alarms - Alarms Generation **** Fuse Locc-Box Current Limit Alarm / **** 2.2 - Alarms - Alarms Generation **** Fuse ETA Current Limit Alarm
   // Memorisation of the Alarm
   IF (#I_AlarmResetPB AND NOT #C_LocalResetCurrentLimit) OR NOT #I_EnableAlarm OR #HMICmdResetCurrentLimit THEN
       #AlarmCurrentLimit := FALSE;   // RS flip-flop
   END_IF;
   IF #AlarmCondCurrentLimit THEN #AlarmCurrentLimit := TRUE; END_IF;
END_REGION

REGION Network 21: **** 2.2 - Alarms - Alarms Generation **** Fuse Locc-Box Current Limit Warning / **** 2.2 - Alarms - Alarms Generation **** Fuse ETA Current Limit Warning
   // Memorisation of the Alarm
   IF (#I_AlarmResetPB AND NOT #C_LocalResetCurrentLimit) OR NOT #I_EnableAlarm OR #HMICmdResetCurrentLimit THEN
       #AD_WarningCurrentLimit := FALSE;   // RS flip-flop
   END_IF;
   IF #FuseNameOK AND #Status.LimitValueCurrent AND #I_EnableAlarm AND NOT #StatusNotAvailable AND #C_LevelCurrentLimit THEN
       #AD_WarningCurrentLimit := TRUE;
   END_IF;
END_REGION

REGION Network 22: **** 2.2 - Alarms - Alarms Generation **** Fuse Locc-Box Under Voltage Alarm (Condtion) / **** 2.2 - Alarms - Alarms Generation **** Fuse ETA Under Voltage Alarm (Condtion)
   // Condition for the Alarm
   #AlarmCondUndVolt := #FuseNameOK AND #Status.LowVoltage AND #I_EnableAlarm AND NOT #StatusNotAvailable AND NOT #C_LevelUndVolt;
END_REGION

REGION Network 23: **** 2.2 - Alarms - Alarms Generation **** Fuse Locc-Box Under Voltage Alarm / **** 2.2 - Alarms - Alarms Generation **** Fuse ETA Under Voltage Alarm
   // Memorisation of the Alarm
   IF (#I_AlarmResetPB AND NOT #C_LocalResetUndVolt) OR NOT #I_EnableAlarm OR #HMICmdResetUndVolt THEN
       #AlarmUndVolt := FALSE;   // RS flip-flop
   END_IF;
   IF #AlarmCondUndVolt THEN #AlarmUndVolt := TRUE; END_IF;
END_REGION

REGION Network 24: **** 2.2 - Alarms - Alarms Generation **** Fuse Locc-Box Under Voltage Warning / **** 2.2 - Alarms - Alarms Generation **** Fuse ETA Under Voltage Warning
   // Memorisation of the Alarm
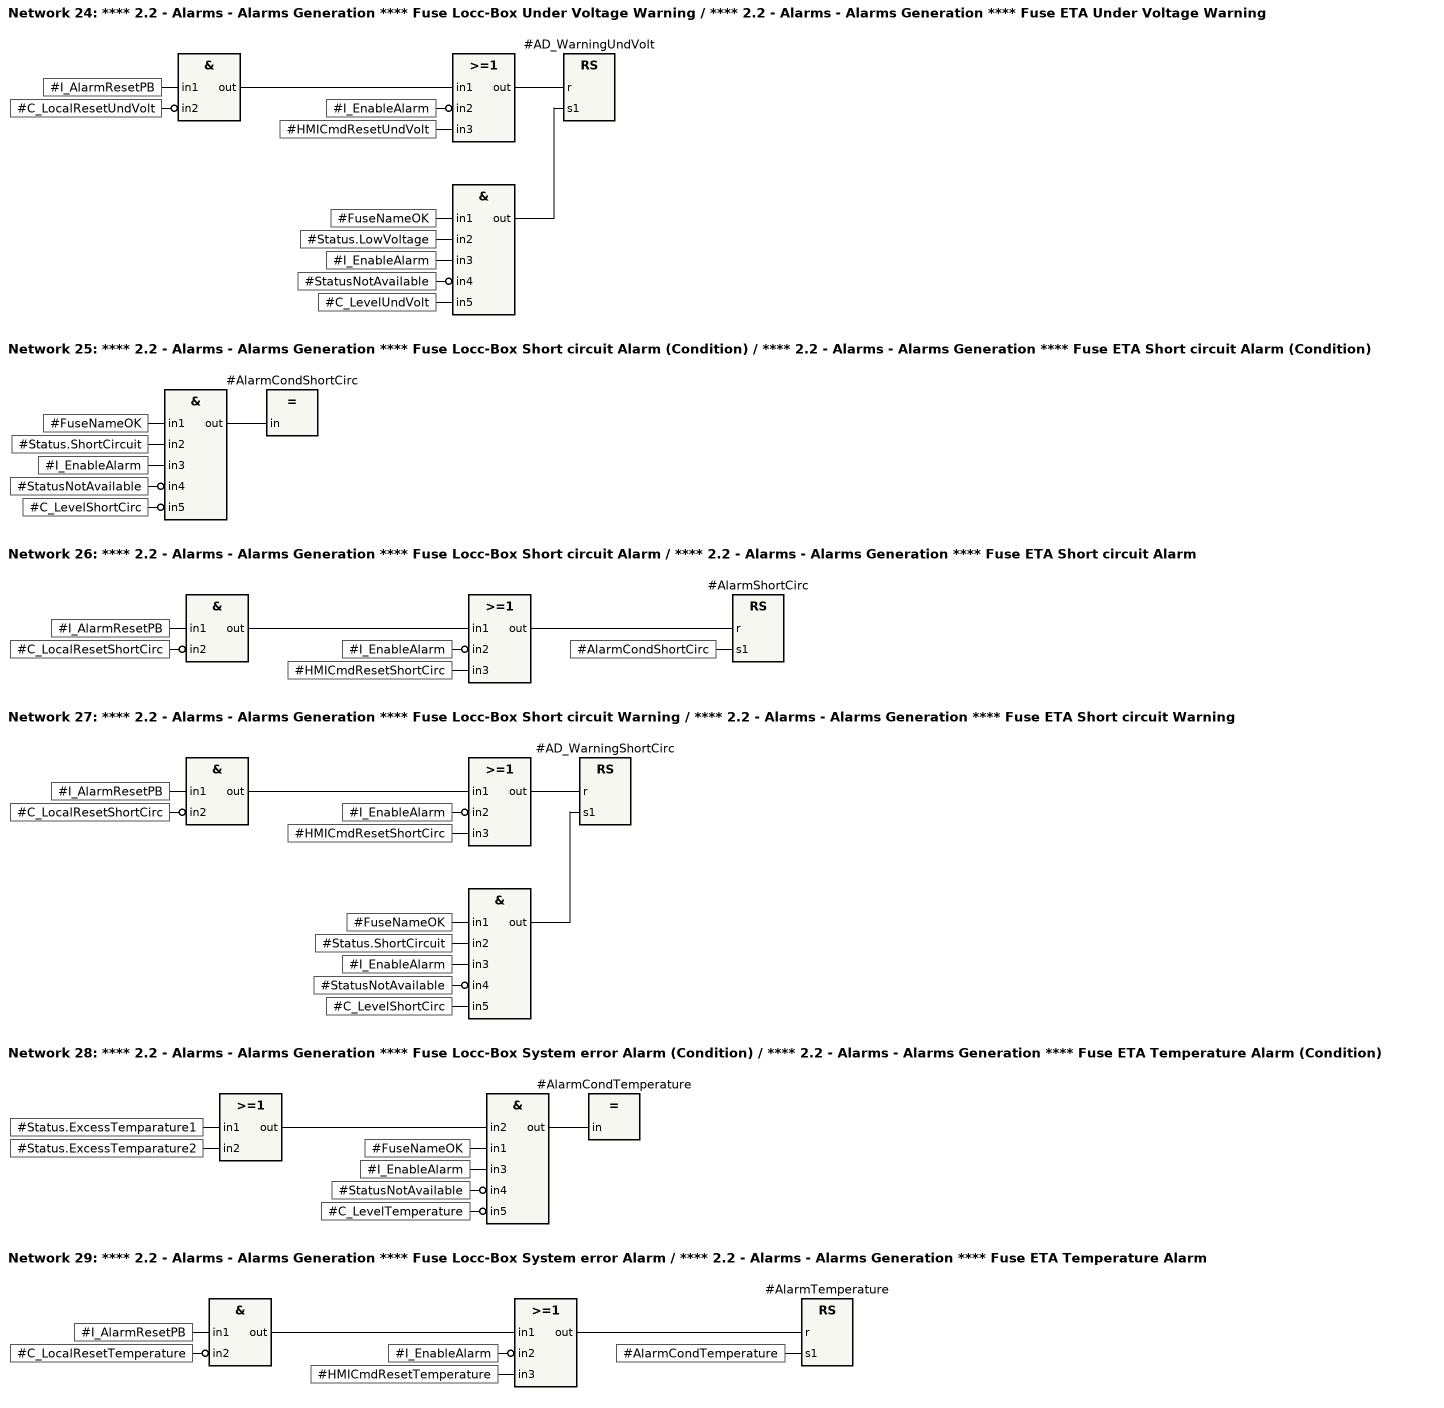
   IF (#I_AlarmResetPB AND NOT #C_LocalResetUndVolt) OR NOT #I_EnableAlarm OR #HMICmdResetUndVolt THEN
       #AD_WarningUndVolt := FALSE;   // RS flip-flop
   END_IF;
   IF #FuseNameOK AND #Status.LowVoltage AND #I_EnableAlarm AND NOT #StatusNotAvailable AND #C_LevelUndVolt THEN
       #AD_WarningUndVolt := TRUE;
   END_IF;
END_REGION

REGION Network 25: **** 2.2 - Alarms - Alarms Generation **** Fuse Locc-Box Short circuit Alarm (Condition) / **** 2.2 - Alarms - Alarms Generation **** Fuse ETA Short circuit Alarm (Condition)
   // Condition for the Alarm
   #AlarmCondShortCirc := #FuseNameOK AND #Status.ShortCircuit AND #I_EnableAlarm AND NOT #StatusNotAvailable AND NOT #C_LevelShortCirc;
END_REGION

REGION Network 26: **** 2.2 - Alarms - Alarms Generation **** Fuse Locc-Box Short circuit Alarm / **** 2.2 - Alarms - Alarms Generation **** Fuse ETA Short circuit Alarm
   // Memorisation of the Alarm
   IF (#I_AlarmResetPB AND NOT #C_LocalResetShortCirc) OR NOT #I_EnableAlarm OR #HMICmdResetShortCirc THEN
       #AlarmShortCirc := FALSE;   // RS flip-flop
   END_IF;
   IF #AlarmCondShortCirc THEN #AlarmShortCirc := TRUE; END_IF;
END_REGION

REGION Network 27: **** 2.2 - Alarms - Alarms Generation **** Fuse Locc-Box Short circuit Warning / **** 2.2 - Alarms - Alarms Generation **** Fuse ETA Short circuit Warning
   // Memorisation of the Alarm
   IF (#I_AlarmResetPB AND NOT #C_LocalResetShortCirc) OR NOT #I_EnableAlarm OR #HMICmdResetShortCirc THEN
       #AD_WarningShortCirc := FALSE;   // RS flip-flop
   END_IF;
   IF #FuseNameOK AND #Status.ShortCircuit AND #I_EnableAlarm AND NOT #StatusNotAvailable AND #C_LevelShortCirc THEN
       #AD_WarningShortCirc := TRUE;
   END_IF;
END_REGION

REGION Network 28: **** 2.2 - Alarms - Alarms Generation **** Fuse Locc-Box System error Alarm (Condition) / **** 2.2 - Alarms - Alarms Generation **** Fuse ETA Temperature Alarm (Condition)
   // Condition for the Alarm
   #AlarmCondTemperature := (#Status.ExcessTemparature1 OR #Status.ExcessTemparature2) AND #FuseNameOK AND #I_EnableAlarm AND NOT #StatusNotAvailable AND NOT #C_LevelTemperature;
END_REGION

REGION Network 29: **** 2.2 - Alarms - Alarms Generation **** Fuse Locc-Box System error Alarm / **** 2.2 - Alarms - Alarms Generation **** Fuse ETA Temperature Alarm
   // Memorisation of the Alarm
   IF (#I_AlarmResetPB AND NOT #C_LocalResetTemperature) OR NOT #I_EnableAlarm OR #HMICmdResetTemperature THEN
       #AlarmTemperature := FALSE;   // RS flip-flop
   END_IF;
   IF #AlarmCondTemperature THEN #AlarmTemperature := TRUE; END_IF;
END_REGION

REGION Network 30: **** 2.2 - Alarms - Alarms Generation **** Fuse Locc-Box System error Warning / **** 2.2 - Alarms - Alarms Generation **** Fuse ETA Temperature Warning
   // Memorisation of the Alarm
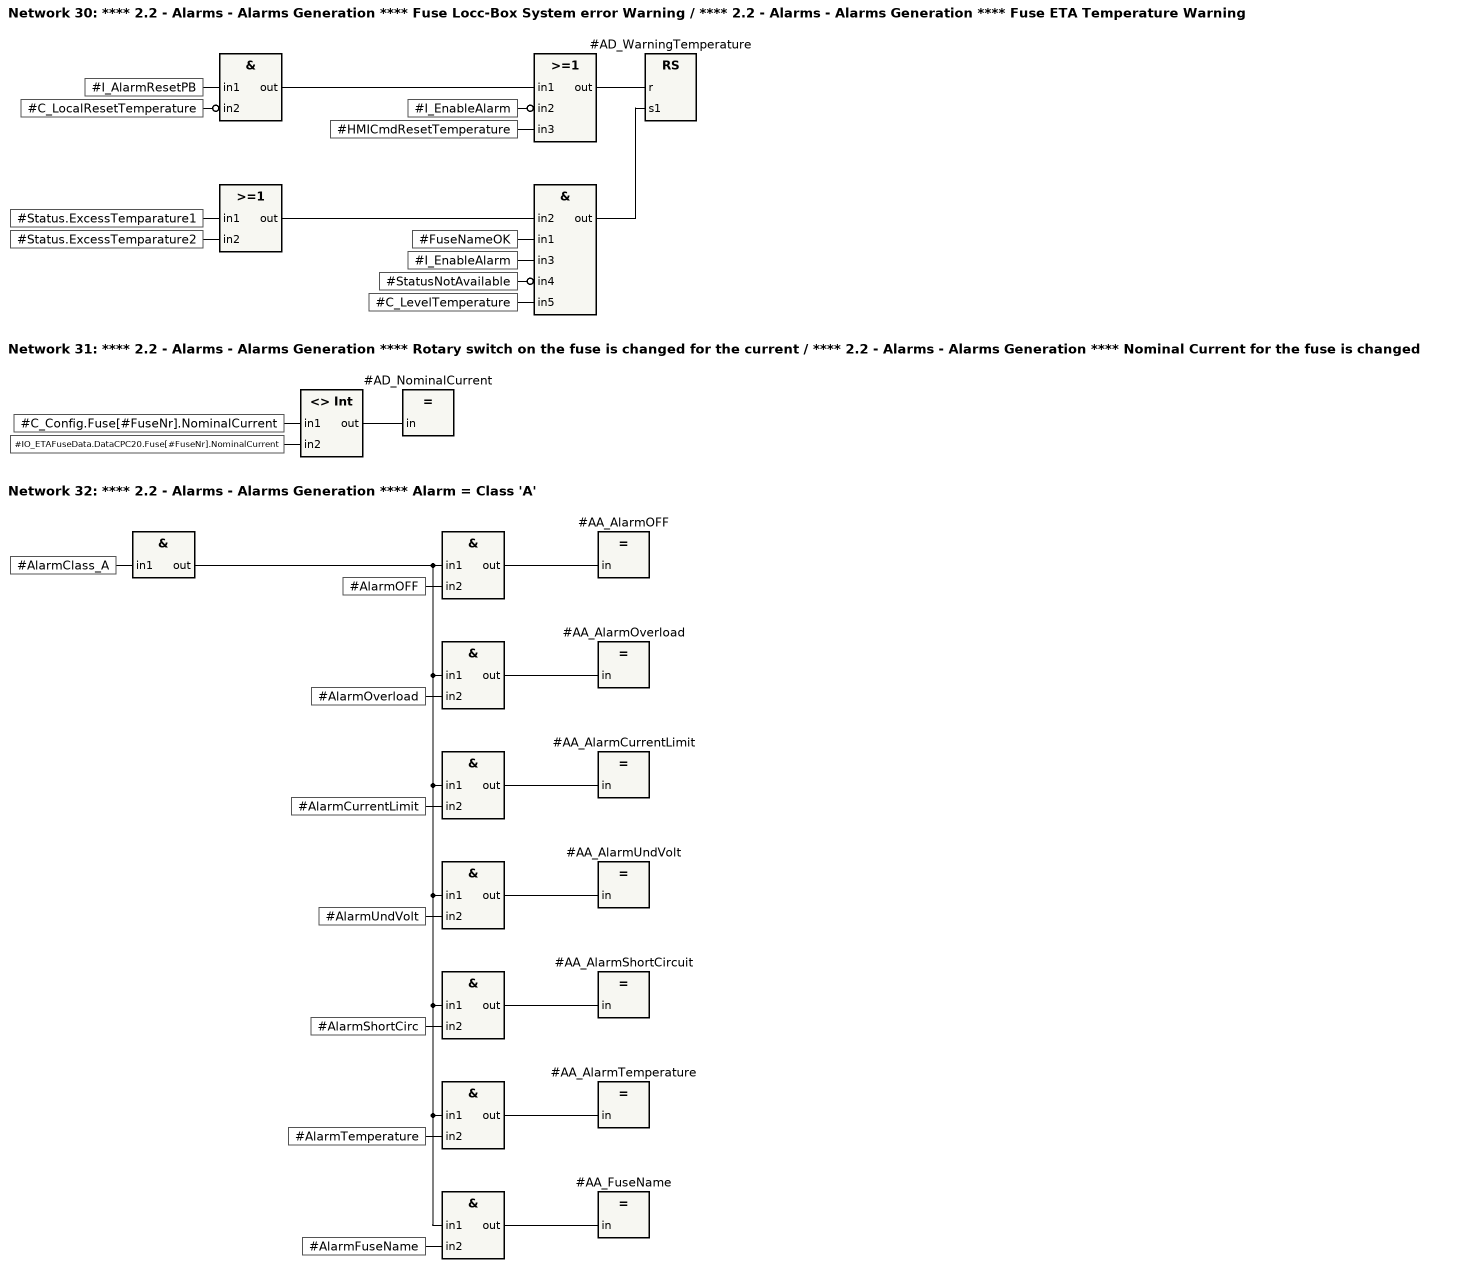
   IF (#I_AlarmResetPB AND NOT #C_LocalResetTemperature) OR NOT #I_EnableAlarm OR #HMICmdResetTemperature THEN
       #AD_WarningTemperature := FALSE;   // RS flip-flop
   END_IF;
   IF (#Status.ExcessTemparature1 OR #Status.ExcessTemparature2) AND #FuseNameOK AND #I_EnableAlarm AND NOT #StatusNotAvailable AND #C_LevelTemperature THEN
       #AD_WarningTemperature := TRUE;
   END_IF;
END_REGION

REGION Network 31: **** 2.2 - Alarms - Alarms Generation **** Rotary switch on the fuse is changed for the current / **** 2.2 - Alarms - Alarms Generation **** Nominal Current for the fuse is changed
   // Alarm
   #AD_NominalCurrent := #C_Config.Fuse[#FuseNr].NominalCurrent <> #IO_ETAFuseData.DataCPC20.Fuse[#FuseNr].NominalCurrent;
END_REGION

REGION Network 32: **** 2.2 - Alarms - Alarms Generation **** Alarm = Class 'A'
   // Alarm = Class 'A'
   #AA_AlarmOFF := #AlarmClass_A AND #AlarmOFF;
   #AA_AlarmOverload := #AlarmClass_A AND #AlarmOverload;
   #AA_AlarmCurrentLimit := #AlarmClass_A AND #AlarmCurrentLimit;
   #AA_AlarmUndVolt := #AlarmClass_A AND #AlarmUndVolt;
   #AA_AlarmShortCircuit := #AlarmClass_A AND #AlarmShortCirc;
   #AA_AlarmTemperature := #AlarmClass_A AND #AlarmTemperature;
   #AA_FuseName := #AlarmClass_A AND #AlarmFuseName;
END_REGION

REGION Network 33: **** 2.2 - Alarms - Alarms Generation **** Alarm = Class 'B'
   // Alarm = Class 'B'
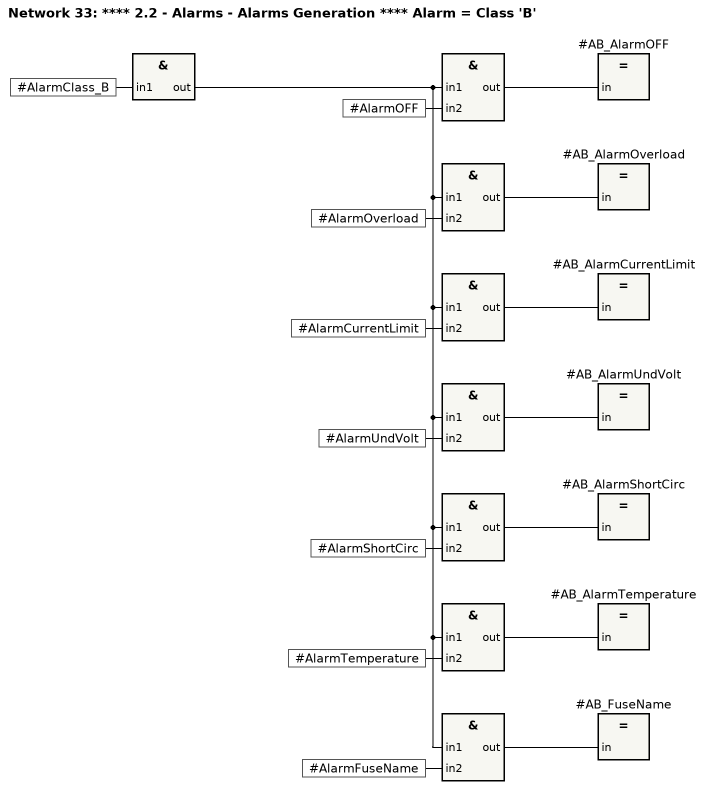
   #AB_AlarmOFF := #AlarmClass_B AND #AlarmOFF;
   #AB_AlarmOverload := #AlarmClass_B AND #AlarmOverload;
   #AB_AlarmCurrentLimit := #AlarmClass_B AND #AlarmCurrentLimit;
   #AB_AlarmUndVolt := #AlarmClass_B AND #AlarmUndVolt;
   #AB_AlarmShortCirc := #AlarmClass_B AND #AlarmShortCirc;
   #AB_AlarmTemperature := #AlarmClass_B AND #AlarmTemperature;
   #AB_FuseName := #AlarmClass_B AND #AlarmFuseName;
END_REGION

REGION Network 34: **** 2.2 - Alarms - Alarms Generation **** Alarm = Class 'C'
   // Alarm = Class 'C'
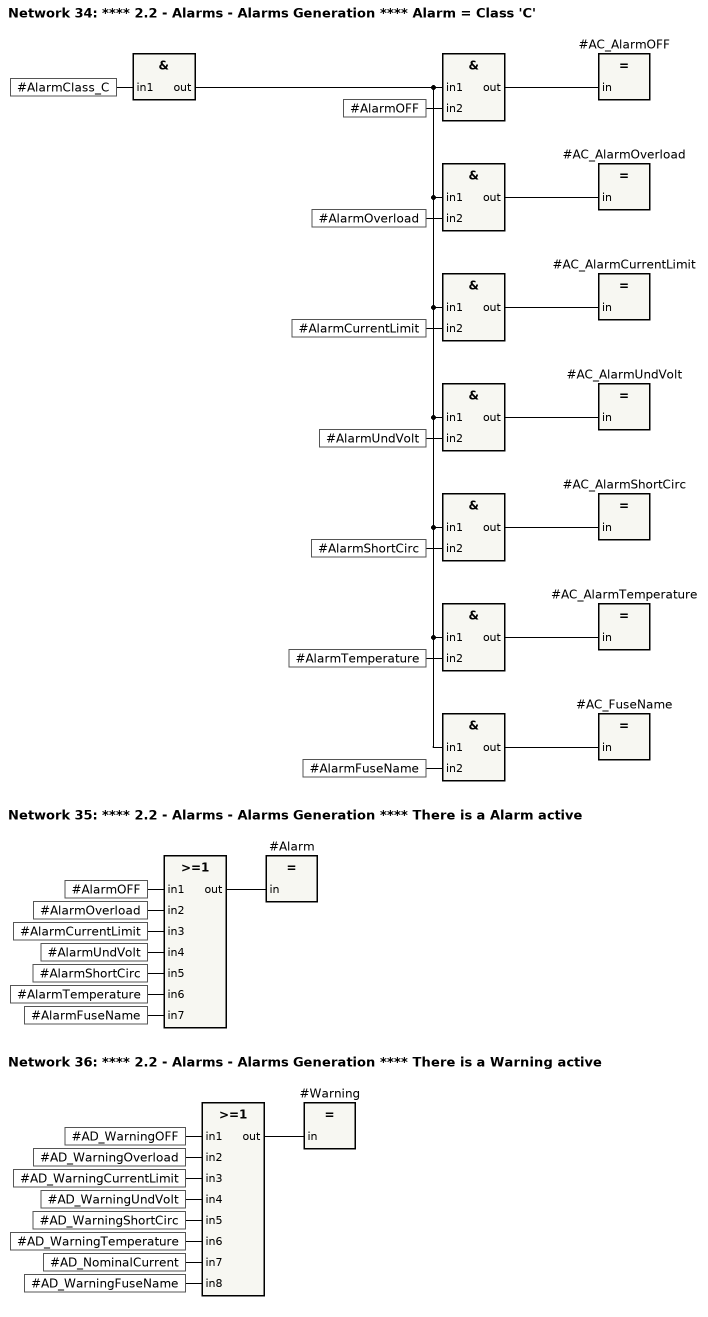
   #AC_AlarmOFF := #AlarmClass_C AND #AlarmOFF;
   #AC_AlarmOverload := #AlarmClass_C AND #AlarmOverload;
   #AC_AlarmCurrentLimit := #AlarmClass_C AND #AlarmCurrentLimit;
   #AC_AlarmUndVolt := #AlarmClass_C AND #AlarmUndVolt;
   #AC_AlarmShortCirc := #AlarmClass_C AND #AlarmShortCirc;
   #AC_AlarmTemperature := #AlarmClass_C AND #AlarmTemperature;
   #AC_FuseName := #AlarmClass_C AND #AlarmFuseName;
END_REGION

REGION Network 35: **** 2.2 - Alarms - Alarms Generation **** There is a Alarm active
   // There is a Alarm active
   #Alarm := #AlarmOFF OR #AlarmOverload OR #AlarmCurrentLimit OR #AlarmUndVolt OR #AlarmShortCirc OR #AlarmTemperature OR #AlarmFuseName;
END_REGION

REGION Network 36: **** 2.2 - Alarms - Alarms Generation **** There is a Warning active
   // There is a Warning active
   #Warning := #AD_WarningOFF OR #AD_WarningOverload OR #AD_WarningCurrentLimit OR #AD_WarningUndVolt OR #AD_WarningShortCirc OR #AD_WarningTemperature OR #AD_NominalCurrent OR #AD_WarningFuseName;
END_REGION

REGION Network 37: **** 4.6 - Mashine Status - Indications **** Icon Animation
   // Icon Animation
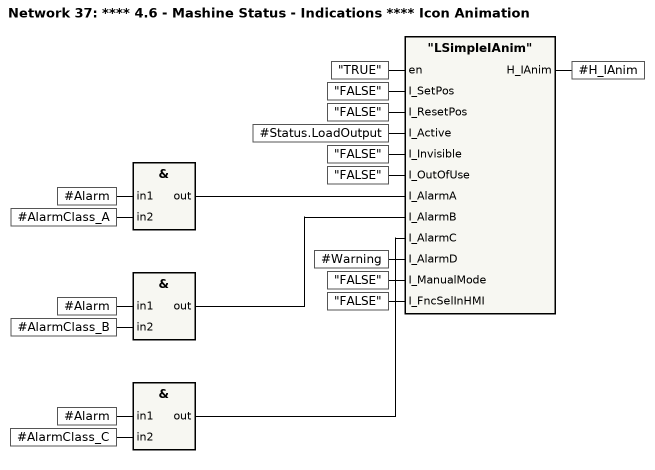
   IF "TRUE" THEN
       "LSimpleIAnim"(I_SetPos := "FALSE",
                      I_ResetPos := "FALSE",
                      I_Active := #Status.LoadOutput,
                      I_Invisible := "FALSE",
                      I_OutOfUse := "FALSE",
                      I_AlarmA := #Alarm AND #AlarmClass_A,
                      I_AlarmB := #Alarm AND #AlarmClass_B,
                      I_AlarmC := #Alarm AND #AlarmClass_C,
                      I_AlarmD := #Warning,
                      I_ManualMode := "FALSE",
                      I_FncSelInHMI := "FALSE",
                      H_IAnim => #H_IAnim);
   END_IF;
END_REGION

REGION Network 38: **** 4.6 - Machine Status - Indications **** Animation
   // Animation
